LIN {X 0,Y 496.38,Z 733.448,A -85,B 0,C 180,E1 23641.747,E2 23641.747} C_VEL
LIN {X 0,Y 498.1,Z 714.982,A -85,B 0,C 180,E1 23640.21,E2 23640.21} C_VEL
LIN {X 0,Y 499.843,Z 694.815,A -85,B 0,C 180,E1 23638.795,E2 23638.795} C_VEL
LIN {X 0,Y 501.44,Z 674.409,A -85,B 0,C 180,E1 23637.63,E2 23637.63} C_VEL
LIN {X 0,Y 502.74,Z 652.978,A -85,B 0,C 180,E1 23636.672,E2 23636.672} C_VEL
LIN {X 0,Y 503.931,Z 629.73,A -85,B 0,C 180,E1 23635.874,E2 23635.874} C_VEL
LIN {X 0,Y 504.846,Z 606.635,A -85,B 0,C 180,E1 23635.308,E2 23635.308} C_VEL
LIN {X 0,Y 505.722,Z 566.306,A -85,B 0,C 180,E1 23634.669,E2 23634.669} C_VEL
LIN {X 0,Y 510.163,Z 554.646,A -85,B 0,C 180,E1 23634.04,E2 23634.04} C_VEL
LIN {X 0,Y 517.035,Z 539.66,A -85,B 0,C 180,E1 23633.305,E2 23633.305} C_VEL
LIN {X 0,Y 524.488,Z 527.632,A -85,B 0,C 180,E1 23632.83,E2 23632.83} C_VEL
LIN {X 0,Y 526.737,Z 523.652,A -85,B 0,C 180,E1 23632.664,E2 23632.664} C_VEL
LIN {X 0,Y 533.302,Z 512.044,A -85,B 0,C 180,E1 23632.187,E2 23632.187} C_VEL
LIN {X 0,Y 542.453,Z 498.435,A -85,B 0,C 180,E1 23631.8,E2 23631.8} C_VEL
LIN {X 0,Y 552.676,Z 482.618,A -85,B 0,C 180,E1 23631.568,E2 23631.568} C_VEL
LIN {X 0,Y 561.127,Z 466.92,A -85,B 0,C 180,E1 23631.466,E2 23631.466} C_VEL
LIN {X 0,Y 567.26,Z 452.489,A -85,B 0,C 180,E1 23631.429,E2 23631.429} C_VEL
LIN {X 0,Y 565.896,Z 454.329,A -85,B 0,C 180,E1 23630.864,E2 23630.864} C_VEL
LIN {X 0,Y 563.058,Z 455.358,A -85,B 0,C 180,E1 23630.255,E2 23630.255} C_VEL
LIN {X 0,Y 559.403,Z 455.291,A -85,B 0,C 180,E1 23629.747,E2 23629.747} C_VEL
LIN {X 0,Y 554.286,Z 453.945,A -85,B 0,C 180,E1 23629.255,E2 23629.255} C_VEL
LIN {X 0,Y 543.774,Z 449.42,A -85,B 0,C 180,E1 23628.29,E2 23628.29} C_VEL
LIN {X 0,Y 534.055,Z 443.361,A -85,B 0,C 180,E1 23627.214,E2 23627.214} C_VEL
LIN {X 0,Y 525.272,Z 435.554,A -85,B 0,C 180,E1 23626.015,E2 23626.015} C_VEL
LIN {X 0,Y 517.9,Z 426.094,A -85,B 0,C 180,E1 23624.727,E2 23624.727} C_VEL
LIN {X 0,Y 512.311,Z 415.203,A -85,B 0,C 180,E1 23623.392,E2 23623.392} C_VEL
LIN {X 0,Y 508.641,Z 403.465,A -85,B 0,C 180,E1 23622.091,E2 23622.091} C_VEL
LIN {X 0,Y 506.405,Z 389.242,A -85,B 0,C 180,E1 23620.659,E2 23620.659} C_VEL
LIN {X 0,Y 505.979,Z 373.52,A -85,B 0,C 180,E1 23619.223,E2 23619.223} C_VEL
LIN {X 0,Y 509.789,Z 322.987,A -85,B 0,C 180,E1 23614.931,E2 23614.931} C_VEL
LIN {X 0,Y 511.824,Z 299.18,A -85,B 0,C 180,E1 23612.833,E2 23612.833} C_VEL
LIN {X 0,Y 504.534,Z 283.166,A -85,B 0,C 180,E1 23610.222,E2 23610.222} C_VEL
LIN {X 0,Y 500.176,Z 274.319,A -85,B 0,C 180,E1 23608.628,E2 23608.628} C_VEL
LIN {X 0,Y 497.624,Z 274.818,A -85,B 0,C 180,E1 23608.306,E2 23608.306} C_VEL
LIN {X 0,Y 495.141,Z 275.99,A -85,B 0,C 180,E1 23608.067,E2 23608.067} C_VEL
LIN {X 0,Y 493.25,Z 276.086,A -85,B 0,C 180,E1 23607.789,E2 23607.789} C_VEL
LIN {X 0,Y 492.541,Z 275.81,A -85,B 0,C 180,E1 23607.619,E2 23607.619} C_VEL
LIN {X 0,Y 493.172,Z 322.85,A -85,B 0,C 180,E1 23604.558,E2 23604.558} C_VEL
LIN {X 0,Y 493.39,Z 364.566,A -85,B 0,C 180,E1 23601.705,E2 23601.705} C_VEL
LIN {X 0,Y 493.167,Z 403.632,A -85,B 0,C 180,E1 23598.928,E2 23598.928} C_VEL
LIN {X 0,Y 492.679,Z 449.513,A -85,B 0,C 180,E1 23595.598,E2 23595.598} C_VEL
LIN {X 0,Y 491.957,Z 495.066,A -85,B 0,C 180,E1 23592.202,E2 23592.202} C_VEL
LIN {X 0,Y 491.446,Z 499.514,A -85,B 0,C 180,E1 23591.926,E2 23591.926} C_VEL
LIN {X 0,Y 490.668,Z 612.915,A -85,B 0,C 180,E1 23590.126,E2 23590.126} C_VEL
LIN {X 0,Y 490.606,Z 628.131,A -85,B 0,C 180,E1 23589.649,E2 23589.649} C_VEL
LIN {X 0,Y 490.477,Z 641.255,A -85,B 0,C 180,E1 23589.031,E2 23589.031} C_VEL
LIN {X 0,Y 490.233,Z 654.167,A -85,B 0,C 180,E1 23588.208,E2 23588.208} C_VEL
LIN {X 0,Y 489.961,Z 666.706,A -85,B 0,C 180,E1 23587.15,E2 23587.15} C_VEL
LIN {X 0,Y 489.656,Z 677.457,A -85,B 0,C 180,E1 23585.977,E2 23585.977} C_VEL
LIN {X 0,Y 489.379,Z 686.759,A -85,B 0,C 180,E1 23584.687,E2 23584.687} C_VEL
LIN {X 0,Y 489.133,Z 694.688,A -85,B 0,C 180,E1 23583.281,E2 23583.281} C_VEL
LIN {X 0,Y 488.904,Z 701.596,A -85,B 0,C 180,E1 23581.64,E2 23581.64} C_VEL
LIN {X 0,Y 488.763,Z 706.452,A -85,B 0,C 180,E1 23580,E2 23580} C_VEL
LIN {X 0,Y 488.665,Z 709.537,A -85,B 0,C 180,E1 23578.358,E2 23578.358} C_VEL
LIN {X 0,Y 488.621,Z 711,A -85,B 0,C 180,E1 23576.598,E2 23576.598} C_VEL
LIN {X 0,Y 488.594,Z 710.599,A -85,B 0,C 180,E1 23574.834,E2 23574.834} C_VEL
LIN {X 0,Y 488.619,Z 708.56,A -85,B 0,C 180,E1 23573.183,E2 23573.183} C_VEL
LIN {X 0,Y 488.682,Z 704.854,A -85,B 0,C 180,E1 23571.528,E2 23571.528} C_VEL
LIN {X 0,Y 488.813,Z 699.231,A -85,B 0,C 180,E1 23569.868,E2 23569.868} C_VEL
LIN {X 0,Y 489.009,Z 692.043,A -85,B 0,C 180,E1 23568.321,E2 23568.321} C_VEL
LIN {X 0,Y 489.261,Z 683.364,A -85,B 0,C 180,E1 23566.888,E2 23566.888} C_VEL
LIN {X 0,Y 489.573,Z 673.151,A -85,B 0,C 180,E1 23565.572,E2 23565.572} C_VEL
LIN {X 0,Y 489.896,Z 661.171,A -85,B 0,C 180,E1 23564.371,E2 23564.371} C_VEL
LIN {X 0,Y 490.193,Z 648.737,A -85,B 0,C 180,E1 23563.407,E2 23563.407} C_VEL
LIN {X 0,Y 490.459,Z 635.31,A -85,B 0,C 180,E1 23562.616,E2 23562.616} C_VEL
LIN {X 0,Y 490.638,Z 620.571,A -85,B 0,C 180,E1 23561.997,E2 23561.997} C_VEL
LIN {X 0,Y 490.728,Z 604.678,A -85,B 0,C 180,E1 23561.586,E2 23561.586} C_VEL
LIN {X 0,Y 491.469,Z 494.156,A -85,B 0,C 180,E1 23559.859,E2 23559.859} C_VEL
LIN {X 0,Y 492.377,Z 448.014,A -85,B 0,C 180,E1 23556.326,E2 23556.326} C_VEL
LIN {X 0,Y 493.343,Z 402.982,A -85,B 0,C 180,E1 23552.87,E2 23552.87} C_VEL
LIN {X 0,Y 494.194,Z 357.923,A -85,B 0,C 180,E1 23549.413,E2 23549.413} C_VEL
LIN {X 0,Y 494.758,Z 323.358,A -85,B 0,C 180,E1 23546.764,E2 23546.764} C_VEL
LIN {X 0,Y 493.985,Z 317.131,A -85,B 0,C 180,E1 23546.234,E2 23546.234} C_VEL
LIN {X 0,Y 488.35,Z 301.373,A -85,B 0,C 180,E1 23544.701,E2 23544.701} C_VEL
LIN {X 0,Y 487.701,Z 295.968,A -85,B 0,C 180,E1 23544.249,E2 23544.249} C_VEL
LIN {X 0,Y 488.094,Z 275.29,A -85,B 0,C 180,E1 23542.639,E2 23542.639} C_VEL
LIN {X 0,Y 480.862,Z 252.836,A -85,B 0,C 180,E1 23540.451,E2 23540.451} C_VEL
LIN {X 0,Y 480.895,Z 253.018,A -85,B 0,C 180,E1 23539.085,E2 23539.085} C_VEL
LIN {X 0,Y 482.364,Z 256.557,A -85,B 0,C 180,E1 23538.265,E2 23538.265} C_VEL
LIN {X 0,Y 483.282,Z 257.796,A -85,B 0,C 180,E1 23537.907,E2 23537.907} C_VEL
LIN {X 0,Y 485.144,Z 261.755,A -85,B 0,C 180,E1 23536.985,E2 23536.985} C_VEL
LIN {X 0,Y 490.291,Z 272.658,A -85,B 0,C 180,E1 23534.55,E2 23534.55} C_VEL
LIN {X 0,Y 495.139,Z 283.311,A -85,B 0,C 180,E1 23532.346,E2 23532.346} C_VEL
LIN {X 0,Y 500.066,Z 295.346,A -85,B 0,C 180,E1 23530.078,E2 23530.078} C_VEL
LIN {X 0,Y 497.632,Z 318.632,A -85,B 0,C 180,E1 23527.59,E2 23527.59} C_VEL
LIN {X 0,Y 498.99,Z 325.374,A -85,B 0,C 180,E1 23527.35,E2 23527.35} C_VEL
LIN {X 0,Y 496.803,Z 427.751,A -85,B 0,C 180,E1 23525.65,E2 23525.65} C_VEL
LIN {X 0,Y 493.178,Z 568.271,A -85,B 0,C 180,E1 23523.126,E2 23523.126} C_VEL
LIN {X 0,Y 492.401,Z 589.199,A -85,B 0,C 180,E1 23522.533,E2 23522.533} C_VEL
LIN {X 0,Y 491.403,Z 608.833,A -85,B 0,C 180,E1 23521.761,E2 23521.761} C_VEL
LIN {X 0,Y 490.219,Z 627.883,A -85,B 0,C 180,E1 23520.794,E2 23520.794} C_VEL
LIN {X 0,Y 488.842,Z 646.705,A -85,B 0,C 180,E1 23519.601,E2 23519.601} C_VEL
LIN {X 0,Y 487.423,Z 664.686,A -85,B 0,C 180,E1 23518.208,E2 23518.208} C_VEL
LIN {X 0,Y 485.977,Z 681.431,A -85,B 0,C 180,E1 23516.649,E2 23516.649} C_VEL
LIN {X 0,Y 484.672,Z 696.234,A -85,B 0,C 180,E1 23515.018,E2 23515.018} C_VEL
LIN {X 0,Y 483.407,Z 710.599,A -85,B 0,C 180,E1 23513.141,E2 23513.141} C_VEL
LIN {X 0,Y 482.297,Z 723.641,A -85,B 0,C 180,E1 23511.106,E2 23511.106} C_VEL
LIN {X 0,Y 481.388,Z 735.453,A -85,B 0,C 180,E1 23508.906,E2 23508.906} C_VEL
LIN {X 0,Y 480.799,Z 744.274,A -85,B 0,C 180,E1 23506.926,E2 23506.926} C_VEL
LIN {X 0,Y 480.356,Z 753.265,A -85,B 0,C 180,E1 23504.588,E2 23504.588} C_VEL
LIN {X 0,Y 480.101,Z 760.219,A -85,B 0,C 180,E1 23502.265,E2 23502.265} C_VEL
LIN {X 0,Y 479.985,Z 765.081,A -85,B 0,C 180,E1 23500.199,E2 23500.199} C_VEL
LIN {X 0,Y 479.931,Z 769.255,A -85,B 0,C 180,E1 23497.783,E2 23497.783} C_VEL
LIN {X 0,Y 479.905,Z 771.524,A -85,B 0,C 180,E1 23495.5,E2 23495.5} C_VEL
LIN {X 0,Y 479.903,Z 772.375,A -85,B 0,C 180,E1 23493.464,E2 23493.464} C_VEL
LIN {X 0,Y 479.907,Z 772.03,A -85,B 0,C 180,E1 23491.194,E2 23491.194} C_VEL
LIN {X 0,Y 479.913,Z 769.901,A -85,B 0,C 180,E1 23488.687,E2 23488.687} C_VEL
LIN {X 0,Y 479.948,Z 766.881,A -85,B 0,C 180,E1 23486.656,E2 23486.656} C_VEL
LIN {X 0,Y 480.034,Z 762.684,A -85,B 0,C 180,E1 23484.622,E2 23484.622} C_VEL
LIN {X 0,Y 480.242,Z 756.178,A -85,B 0,C 180,E1 23482.222,E2 23482.222} C_VEL
LIN {X 0,Y 480.57,Z 748.581,A -85,B 0,C 180,E1 23480.056,E2 23480.056} C_VEL
LIN {X 0,Y 481.199,Z 738.233,A -85,B 0,C 180,E1 23477.58,E2 23477.58} C_VEL
LIN {X 0,Y 481.993,Z 727.382,A -85,B 0,C 180,E1 23475.463,E2 23475.463} C_VEL
LIN {X 0,Y 483.026,Z 714.869,A -85,B 0,C 180,E1 23473.402,E2 23473.402} C_VEL
LIN {X 0,Y 484.264,Z 700.8,A -85,B 0,C 180,E1 23471.46,E2 23471.46} C_VEL
LIN {X 0,Y 485.557,Z 686.249,A -85,B 0,C 180,E1 23469.76,E2 23469.76} C_VEL
LIN {X 0,Y 487.016,Z 669.572,A -85,B 0,C 180,E1 23468.122,E2 23468.122} C_VEL
LIN {X 0,Y 488.472,Z 651.962,A -85,B 0,C 180,E1 23466.683,E2 23466.683} C_VEL
LIN {X 0,Y 489.911,Z 632.774,A -85,B 0,C 180,E1 23465.396,E2 23465.396} C_VEL
LIN {X 0,Y 491.095,Z 614.617,A -85,B 0,C 180,E1 23464.415,E2 23464.415} C_VEL
LIN {X 0,Y 492.12,Z 595.098,A -85,B 0,C 180,E1 23463.584,E2 23463.584} C_VEL
LIN {X 0,Y 492.975,Z 574.762,A -85,B 0,C 180,E1 23462.943,E2 23462.943} C_VEL
LIN {X 0,Y 493.591,Z 552.537,A -85,B 0,C 180,E1 23462.471,E2 23462.471} C_VEL
LIN {X 0,Y 497.835,Z 385.617,A -85,B 0,C 180,E1 23459.542,E2 23459.542} C_VEL
LIN {X 0,Y 498.921,Z 320.717,A -85,B 0,C 180,E1 23458.474,E2 23458.474} C_VEL
LIN {X 0,Y 498.1,Z 316.099,A -85,B 0,C 180,E1 23458.303,E2 23458.303} C_VEL
LIN {X 0,Y 500.032,Z 293.482,A -85,B 0,C 180,E1 23456.288,E2 23456.288} C_VEL
LIN {X 0,Y 492.25,Z 276.567,A -85,B 0,C 180,E1 23453.549,E2 23453.549} C_VEL
LIN {X 0,Y 486.502,Z 264.754,A -85,B 0,C 180,E1 23451.484,E2 23451.484} C_VEL
LIN {X 0,Y 484.789,Z 261.244,A -85,B 0,C 180,E1 23450.85,E2 23450.85} C_VEL
LIN {X 0,Y 482.59,Z 256.865,A -85,B 0,C 180,E1 23450.038,E2 23450.038} C_VEL
LIN {X 0,Y 480.993,Z 253.436,A -85,B 0,C 180,E1 23449.409,E2 23449.409} C_VEL
LIN {X 0,Y 480.894,Z 252.838,A -85,B 0,C 180,E1 23449.321,E2 23449.321} C_VEL
LIN {X 0,Y 480.885,Z 252.835,A -85,B 0,C 180,E1 23445.664,E2 23445.664} C_VEL
LIN {X 0,Y 480.883,Z 252.833,A -85,B 0,C 180,E1 23442.03,E2 23442.03} C_VEL
LIN {X 0,Y 480.896,Z 252.833,A -85,B 0,C 180,E1 23438.386,E2 23438.386} C_VEL
LIN {X 0,Y 480.882,Z 252.837,A -85,B 0,C 180,E1 23434.73,E2 23434.73} C_VEL
LIN {X 0,Y 480.882,Z 252.884,A -85,B 0,C 180,E1 23431.161,E2 23431.161} C_VEL
LIN {X 0,Y 488.38,Z 276.554,A -85,B 0,C 180,E1 23428.692,E2 23428.692} C_VEL
LIN {X 0,Y 487.688,Z 321.036,A -85,B 0,C 180,E1 23424.983,E2 23424.983} C_VEL
LIN {X 0,Y 486.877,Z 362.038,A -85,B 0,C 180,E1 23421.568,E2 23421.568} C_VEL
LIN {X 0,Y 485.897,Z 404.107,A -85,B 0,C 180,E1 23418.067,E2 23418.067} C_VEL
LIN {X 0,Y 484.975,Z 446.252,A -85,B 0,C 180,E1 23414.587,E2 23414.587} C_VEL
LIN {X 0,Y 485.216,Z 454.797,A -85,B 0,C 180,E1 23414.435,E2 23414.435} C_VEL
LIN {X 0,Y 483.933,Z 589.379,A -85,B 0,C 180,E1 23412.267,E2 23412.267} C_VEL
LIN {X 0,Y 483.783,Z 605.964,A -85,B 0,C 180,E1 23411.777,E2 23411.777} C_VEL
LIN {X 0,Y 483.477,Z 621.487,A -85,B 0,C 180,E1 23411.089,E2 23411.089} C_VEL
LIN {X 0,Y 483.104,Z 636.557,A -85,B 0,C 180,E1 23410.193,E2 23410.193} C_VEL
LIN {X 0,Y 482.632,Z 651.077,A -85,B 0,C 180,E1 23409.059,E2 23409.059} C_VEL
LIN {X 0,Y 482.198,Z 663.25,A -85,B 0,C 180,E1 23407.866,E2 23407.866} C_VEL
LIN {X 0,Y 481.749,Z 674.924,A -85,B 0,C 180,E1 23406.435,E2 23406.435} C_VEL
LIN {X 0,Y 481.367,Z 685.044,A -85,B 0,C 180,E1 23404.886,E2 23404.886} C_VEL
LIN {X 0,Y 481.07,Z 693.633,A -85,B 0,C 180,E1 23403.217,E2 23403.217} C_VEL
LIN {X 0,Y 480.885,Z 700.29,A -85,B 0,C 180,E1 23401.549,E2 23401.549} C_VEL
LIN {X 0,Y 480.74,Z 705.866,A -85,B 0,C 180,E1 23399.643,E2 23399.643} C_VEL
LIN {X 0,Y 480.686,Z 709.337,A -85,B 0,C 180,E1 23397.855,E2 23397.855} C_VEL
LIN {X 0,Y 480.667,Z 711.381,A -85,B 0,C 180,E1 23395.825,E2 23395.825} C_VEL
LIN {X 0,Y 480.706,Z 711.456,A -85,B 0,C 180,E1 23393.911,E2 23393.911} C_VEL
LIN {X 0,Y 480.777,Z 709.805,A -85,B 0,C 180,E1 23391.991,E2 23391.991} C_VEL
LIN {X 0,Y 480.905,Z 706.23,A -85,B 0,C 180,E1 23390.063,E2 23390.063} C_VEL
LIN {X 0,Y 481.093,Z 701.074,A -85,B 0,C 180,E1 23388.249,E2 23388.249} C_VEL
LIN {X 0,Y 481.341,Z 693.803,A -85,B 0,C 180,E1 23386.425,E2 23386.425} C_VEL
LIN {X 0,Y 481.666,Z 685.525,A -85,B 0,C 180,E1 23384.838,E2 23384.838} C_VEL
LIN {X 0,Y 482.074,Z 674.914,A -85,B 0,C 180,E1 23383.244,E2 23383.244} C_VEL
LIN {X 0,Y 482.486,Z 663.45,A -85,B 0,C 180,E1 23381.89,E2 23381.89} C_VEL
LIN {X 0,Y 482.88,Z 651.01,A -85,B 0,C 180,E1 23380.716,E2 23380.716} C_VEL
LIN {X 0,Y 483.211,Z 637.613,A -85,B 0,C 180,E1 23379.721,E2 23379.721} C_VEL
LIN {X 0,Y 483.487,Z 622.444,A -85,B 0,C 180,E1 23378.857,E2 23378.857} C_VEL
LIN {X 0,Y 483.652,Z 606.109,A -85,B 0,C 180,E1 23378.197,E2 23378.197} C_VEL
LIN {X 0,Y 483.672,Z 589.924,A -85,B 0,C 180,E1 23377.774,E2 23377.774} C_VEL
LIN {X 0,Y 484.709,Z 473.284,A -85,B 0,C 180,E1 23375.896,E2 23375.896} C_VEL
LIN {X 0,Y 485.05,Z 452.809,A -85,B 0,C 180,E1 23375.523,E2 23375.523} C_VEL
LIN {X 0,Y 485.709,Z 447.24,A -85,B 0,C 180,E1 23375.104,E2 23375.104} C_VEL
LIN {X 0,Y 486.235,Z 406.579,A -85,B 0,C 180,E1 23371.906,E2 23371.906} C_VEL
LIN {X 0,Y 486.403,Z 373.966,A -85,B 0,C 180,E1 23369.426,E2 23369.426} C_VEL
LIN {X 0,Y 486.241,Z 335.387,A -85,B 0,C 180,E1 23366.602,E2 23366.602} C_VEL
LIN {X 0,Y 486.068,Z 315.437,A -85,B 0,C 180,E1 23365.175,E2 23365.175} C_VEL
LIN {X 0,Y 487.432,Z 316.242,A -85,B 0,C 180,E1 23364.946,E2 23364.946} C_VEL
LIN {X 0,Y 489.679,Z 316.055,A -85,B 0,C 180,E1 23364.701,E2 23364.701} C_VEL
LIN {X 0,Y 491.846,Z 315.218,A -85,B 0,C 180,E1 23364.523,E2 23364.523} C_VEL
LIN {X 0,Y 495.198,Z 315.029,A -85,B 0,C 180,E1 23364.159,E2 23364.159} C_VEL
LIN {X 0,Y 498.446,Z 314.267,A -85,B 0,C 180,E1 23363.861,E2 23363.861} C_VEL
LIN {X 0,Y 503.576,Z 313.442,A -85,B 0,C 180,E1 23363.37,E2 23363.37} C_VEL
LIN {X 0,Y 502.225,Z 340.421,A -85,B 0,C 180,E1 23361.382,E2 23361.382} C_VEL
LIN {X 0,Y 503.133,Z 357.34,A -85,B 0,C 180,E1 23359.994,E2 23359.994} C_VEL
LIN {X 0,Y 505.646,Z 371.909,A -85,B 0,C 180,E1 23358.666,E2 23358.666} C_VEL
LIN {X 0,Y 509.605,Z 384.438,A -85,B 0,C 180,E1 23357.399,E2 23357.399} C_VEL
LIN {X 0,Y 515.13,Z 395.571,A -85,B 0,C 180,E1 23356.138,E2 23356.138} C_VEL
LIN {X 0,Y 522.184,Z 405.312,A -85,B 0,C 180,E1 23354.891,E2 23354.891} C_VEL
LIN {X 0,Y 530.1,Z 413.14,A -85,B 0,C 180,E1 23353.747,E2 23353.747} C_VEL
LIN {X 0,Y 540.174,Z 420.213,A -85,B 0,C 180,E1 23352.55,E2 23352.55} C_VEL
LIN {X 0,Y 551.135,Z 425.486,A -85,B 0,C 180,E1 23351.466,E2 23351.466} C_VEL
LIN {X 0,Y 560.238,Z 428.38,A -85,B 0,C 180,E1 23350.668,E2 23350.668} C_VEL
LIN {X 0,Y 564.412,Z 428.784,A -85,B 0,C 180,E1 23350.153,E2 23350.153} C_VEL
LIN {X 0,Y 566.541,Z 428.672,A -85,B 0,C 180,E1 23349.758,E2 23349.758} C_VEL
LIN {X 0,Y 564.158,Z 434.639,A -85,B 0,C 180,E1 23349.612,E2 23349.612} C_VEL
LIN {X 0,Y 554.295,Z 452.798,A -85,B 0,C 180,E1 23349.463,E2 23349.463} C_VEL
LIN {X 0,Y 542.754,Z 471.192,A -85,B 0,C 180,E1 23349.144,E2 23349.144} C_VEL
LIN {X 0,Y 529.479,Z 492.499,A -85,B 0,C 180,E1 23348.617,E2 23348.617} C_VEL
LIN {X 0,Y 521.442,Z 507.86,A -85,B 0,C 180,E1 23348.129,E2 23348.129} C_VEL
LIN {X 0,Y 516.353,Z 520.01,A -85,B 0,C 180,E1 23347.657,E2 23347.657} C_VEL
LIN {X 0,Y 509.506,Z 533.706,A -85,B 0,C 180,E1 23347.181,E2 23347.181} C_VEL
LIN {X 0,Y 504.963,Z 545.921,A -85,B 0,C 180,E1 23346.655,E2 23346.655} C_VEL
LIN {X 0,Y 500.019,Z 560.23,A -85,B 0,C 180,E1 23346.008,E2 23346.008} C_VEL
LIN {X 0,Y 499.1,Z 563.948,A -85,B 0,C 180,E1 23345.861,E2 23345.861} C_VEL
LIN {X 0,Y 498.399,Z 593.728,A -85,B 0,C 180,E1 23345.409,E2 23345.409} C_VEL
LIN {X 0,Y 497.549,Z 617.702,A -85,B 0,C 180,E1 23344.92,E2 23344.92} C_VEL
LIN {X 0,Y 496.401,Z 640.592,A -85,B 0,C 180,E1 23344.236,E2 23344.236} C_VEL
LIN {X 0,Y 495.064,Z 662.664,A -85,B 0,C 180,E1 23343.357,E2 23343.357} C_VEL
LIN {X 0,Y 493.532,Z 684.32,A -85,B 0,C 180,E1 23342.265,E2 23342.265} C_VEL
LIN {X 0,Y 491.889,Z 704.756,A -85,B 0,C 180,E1 23340.997,E2 23340.997} C_VEL
LIN {X 0,Y 490.417,Z 721.095,A -85,B 0,C 180,E1 23339.783,E2 23339.783} C_VEL
LIN {X 0,Y 488.503,Z 740.079,A -85,B 0,C 180,E1 23338.084,E2 23338.084} C_VEL
LIN {X 0,Y 486.678,Z 757.864,A -85,B 0,C 180,E1 23336.213,E2 23336.213} C_VEL
LIN {X 0,Y 484.943,Z 774.948,A -85,B 0,C 180,E1 23334.094,E2 23334.094} C_VEL
LIN {X 0,Y 483.4,Z 791.073,A -85,B 0,C 180,E1 23331.731,E2 23331.731} C_VEL
LIN {X 0,Y 482.171,Z 805.314,A -85,B 0,C 180,E1 23329.251,E2 23329.251} C_VEL
LIN {X 0,Y 481.256,Z 817.549,A -85,B 0,C 180,E1 23326.711,E2 23326.711} C_VEL
LIN {X 0,Y 480.623,Z 827.996,A -85,B 0,C 180,E1 23324.087,E2 23324.087} C_VEL
LIN {X 0,Y 480.228,Z 836.573,A -85,B 0,C 180,E1 23321.408,E2 23321.408} C_VEL
LIN {X 0,Y 480.015,Z 843.196,A -85,B 0,C 180,E1 23318.746,E2 23318.746} C_VEL
LIN {X 0,Y 479.938,Z 847.807,A -85,B 0,C 180,E1 23316.219,E2 23316.219} C_VEL
LIN {X 0,Y 479.909,Z 850.87,A -85,B 0,C 180,E1 23313.661,E2 23313.661} C_VEL
LIN {X 0,Y 479.91,Z 852.372,A -85,B 0,C 180,E1 23310.955,E2 23310.955} C_VEL
LIN {X 0,Y 479.899,Z 852.152,A -85,B 0,C 180,E1 23308.328,E2 23308.328} C_VEL
LIN {X 0,Y 479.915,Z 850.371,A -85,B 0,C 180,E1 23305.818,E2 23305.818} C_VEL
LIN {X 0,Y 479.957,Z 846.849,A -85,B 0,C 180,E1 23303.18,E2 23303.18} C_VEL
LIN {X 0,Y 480.072,Z 841.593,A -85,B 0,C 180,E1 23300.53,E2 23300.53} C_VEL
LIN {X 0,Y 480.31,Z 834.427,A -85,B 0,C 180,E1 23297.863,E2 23297.863} C_VEL
LIN {X 0,Y 480.752,Z 825.57,A -85,B 0,C 180,E1 23295.261,E2 23295.261} C_VEL
LIN {X 0,Y 481.437,Z 815,A -85,B 0,C 180,E1 23292.723,E2 23292.723} C_VEL
LIN {X 0,Y 482.332,Z 803.331,A -85,B 0,C 180,E1 23290.377,E2 23290.377} C_VEL
LIN {X 0,Y 483.473,Z 790.295,A -85,B 0,C 180,E1 23288.145,E2 23288.145} C_VEL
LIN {X 0,Y 484.988,Z 774.48,A -85,B 0,C 180,E1 23285.843,E2 23285.843} C_VEL
LIN {X 0,Y 486.71,Z 757.504,A -85,B 0,C 180,E1 23283.746,E2 23283.746} C_VEL
LIN {X 0,Y 488.565,Z 739.511,A -85,B 0,C 180,E1 23281.86,E2 23281.86} C_VEL
LIN {X 0,Y 490.417,Z 721.096,A -85,B 0,C 180,E1 23280.217,E2 23280.217} C_VEL
LIN {X 0,Y 491.89,Z 704.76,A -85,B 0,C 180,E1 23279.003,E2 23279.003} C_VEL
LIN {X 0,Y 493.523,Z 684.24,A -85,B 0,C 180,E1 23277.734,E2 23277.734} C_VEL
LIN {X 0,Y 495.105,Z 661.858,A -85,B 0,C 180,E1 23276.611,E2 23276.611} C_VEL
LIN {X 0,Y 496.481,Z 638.809,A -85,B 0,C 180,E1 23275.705,E2 23275.705} C_VEL
LIN {X 0,Y 497.615,Z 615.774,A -85,B 0,C 180,E1 23275.04,E2 23275.04} C_VEL
LIN {X 0,Y 498.381,Z 592.976,A -85,B 0,C 180,E1 23274.585,E2 23274.585} C_VEL
LIN {X 0,Y 499.034,Z 565.629,A -85,B 0,C 180,E1 23274.171,E2 23274.171} C_VEL
LIN {X 0,Y 499.312,Z 563.71,A -85,B 0,C 180,E1 23274.145,E2 23274.145} C_VEL
LIN {X 0,Y 503.862,Z 552.303,A -85,B 0,C 180,E1 23273.535,E2 23273.535} C_VEL
LIN {X 0,Y 510.541,Z 537.864,A -85,B 0,C 180,E1 23272.824,E2 23272.824} C_VEL
LIN {X 0,Y 517.954,Z 525.867,A -85,B 0,C 180,E1 23272.347,E2 23272.347} C_VEL
LIN {X 0,Y 520.245,Z 521.945,A -85,B 0,C 180,E1 23272.187,E2 23272.187} C_VEL
LIN {X 0,Y 526.825,Z 510.336,A -85,B 0,C 180,E1 23271.708,E2 23271.708} C_VEL
LIN {X 0,Y 536.729,Z 496.264,A -85,B 0,C 180,E1 23271.249,E2 23271.249} C_VEL
LIN {X 0,Y 549.126,Z 480.047,A -85,B 0,C 180,E1 23270.865,E2 23270.865} C_VEL
LIN {X 0,Y 559.176,Z 465.05,A -85,B 0,C 180,E1 23270.688,E2 23270.688} C_VEL
LIN {X 0,Y 560.818,Z 462.177,A -85,B 0,C 180,E1 23270.652,E2 23270.652} C_VEL
LIN {X 0,Y 556.708,Z 462.22,A -85,B 0,C 180,E1 23270.076,E2 23270.076} C_VEL
LIN {X 0,Y 551.539,Z 460.939,A -85,B 0,C 180,E1 23269.587,E2 23269.587} C_VEL
LIN {X 0,Y 540.155,Z 456.256,A -85,B 0,C 180,E1 23268.562,E2 23268.562} C_VEL
LIN {X 0,Y 529.628,Z 449.931,A -85,B 0,C 180,E1 23267.414,E2 23267.414} C_VEL
LIN {X 0,Y 520.709,Z 442.355,A -85,B 0,C 180,E1 23266.219,E2 23266.219} C_VEL
LIN {X 0,Y 512.885,Z 432.876,A -85,B 0,C 180,E1 23264.887,E2 23264.887} C_VEL
LIN {X 0,Y 507.27,Z 422.944,A -85,B 0,C 180,E1 23263.619,E2 23263.619} C_VEL
LIN {X 0,Y 503.046,Z 411.454,A -85,B 0,C 180,E1 23262.284,E2 23262.284} C_VEL
LIN {X 0,Y 500.267,Z 397.472,A -85,B 0,C 180,E1 23260.81,E2 23260.81} C_VEL
LIN {X 0,Y 499.292,Z 382.036,A -85,B 0,C 180,E1 23259.331,E2 23259.331} C_VEL
LIN {X 0,Y 500.645,Z 357.876,A -85,B 0,C 180,E1 23257.238,E2 23257.238} C_VEL
LIN {X 0,Y 504.106,Z 318.983,A -85,B 0,C 180,E1 23253.872,E2 23253.872} C_VEL
LIN {X 0,Y 505.57,Z 303.35,A -85,B 0,C 180,E1 23252.475,E2 23252.475} C_VEL
LIN {X 0,Y 498.672,Z 288.161,A -85,B 0,C 180,E1 23249.95,E2 23249.95} C_VEL
LIN {X 0,Y 495.465,Z 281.71,A -85,B 0,C 180,E1 23248.77,E2 23248.77} C_VEL
LIN {X 0,Y 492.031,Z 282.889,A -85,B 0,C 180,E1 23248.392,E2 23248.392} C_VEL
LIN {X 0,Y 490.315,Z 283.206,A -85,B 0,C 180,E1 23248.169,E2 23248.169} C_VEL
LIN {X 0,Y 487.449,Z 284.527,A -85,B 0,C 180,E1 23247.883,E2 23247.883} C_VEL
LIN {X 0,Y 485.632,Z 284.494,A -85,B 0,C 180,E1 23247.596,E2 23247.596} C_VEL
LIN {X 0,Y 485.142,Z 284.235,A -85,B 0,C 180,E1 23247.477,E2 23247.477} C_VEL
LIN {X 0,Y 485.749,Z 328.431,A -85,B 0,C 180,E1 23244.569,E2 23244.569} C_VEL
LIN {X 0,Y 485.861,Z 371.281,A -85,B 0,C 180,E1 23241.614,E2 23241.614} C_VEL
LIN {X 0,Y 485.548,Z 419.344,A -85,B 0,C 180,E1 23238.178,E2 23238.178} C_VEL
LIN {X 0,Y 484.87,Z 466.154,A -85,B 0,C 180,E1 23234.728,E2 23234.728} C_VEL
LIN {X 0,Y 484.263,Z 497.232,A -85,B 0,C 180,E1 23232.399,E2 23232.399} C_VEL
LIN {X 0,Y 483.749,Z 501.19,A -85,B 0,C 180,E1 23232.163,E2 23232.163} C_VEL
LIN {X 0,Y 482.895,Z 614.459,A -85,B 0,C 180,E1 23230.317,E2 23230.317} C_VEL
LIN {X 0,Y 482.846,Z 629.57,A -85,B 0,C 180,E1 23229.836,E2 23229.836} C_VEL
LIN {X 0,Y 482.707,Z 643.257,A -85,B 0,C 180,E1 23229.177,E2 23229.177} C_VEL
LIN {X 0,Y 482.451,Z 656.435,A -85,B 0,C 180,E1 23228.31,E2 23228.31} C_VEL
LIN {X 0,Y 482.174,Z 668.503,A -85,B 0,C 180,E1 23227.267,E2 23227.267} C_VEL
LIN {X 0,Y 481.827,Z 680.148,A -85,B 0,C 180,E1 23225.955,E2 23225.955} C_VEL
LIN {X 0,Y 481.511,Z 689.887,A -85,B 0,C 180,E1 23224.525,E2 23224.525} C_VEL
LIN {X 0,Y 481.242,Z 697.391,A -85,B 0,C 180,E1 23223.096,E2 23223.096} C_VEL
LIN {X 0,Y 481.035,Z 703.565,A -85,B 0,C 180,E1 23221.548,E2 23221.548} C_VEL
LIN {X 0,Y 480.871,Z 708.507,A -85,B 0,C 180,E1 23219.761,E2 23219.761} C_VEL
LIN {X 0,Y 480.773,Z 711.389,A -85,B 0,C 180,E1 23217.973,E2 23217.973} C_VEL
LIN {X 0,Y 480.717,Z 712.383,A -85,B 0,C 180,E1 23216.183,E2 23216.183} C_VEL
LIN {X 0,Y 480.706,Z 711.653,A -85,B 0,C 180,E1 23214.509,E2 23214.509} C_VEL
LIN {X 0,Y 480.743,Z 709.057,A -85,B 0,C 180,E1 23212.711,E2 23212.711} C_VEL
LIN {X 0,Y 480.838,Z 704.447,A -85,B 0,C 180,E1 23210.907,E2 23210.907} C_VEL
LIN {X 0,Y 481.004,Z 698.083,A -85,B 0,C 180,E1 23209.217,E2 23209.217} C_VEL
LIN {X 0,Y 481.224,Z 690.77,A -85,B 0,C 180,E1 23207.764,E2 23207.764} C_VEL
LIN {X 0,Y 481.525,Z 681.309,A -85,B 0,C 180,E1 23206.307,E2 23206.307} C_VEL
LIN {X 0,Y 481.869,Z 670.1,A -85,B 0,C 180,E1 23204.967,E2 23204.967} C_VEL
LIN {X 0,Y 482.211,Z 657.531,A -85,B 0,C 180,E1 23203.806,E2 23203.806} C_VEL
LIN {X 0,Y 482.547,Z 643.518,A -85,B 0,C 180,E1 23202.826,E2 23202.826} C_VEL
LIN {X 0,Y 482.772,Z 629.023,A -85,B 0,C 180,E1 23202.089,E2 23202.089} C_VEL
LIN {X 0,Y 482.902,Z 614.383,A -85,B 0,C 180,E1 23201.585,E2 23201.585} C_VEL
LIN {X 0,Y 482.941,Z 597.395,A -85,B 0,C 180,E1 23201.255,E2 23201.255} C_VEL
LIN {X 0,Y 483.8,Z 495.19,A -85,B 0,C 180,E1 23199.62,E2 23199.62} C_VEL
LIN {X 0,Y 484.747,Z 449.326,A -85,B 0,C 180,E1 23196.089,E2 23196.089} C_VEL
LIN {X 0,Y 485.741,Z 405.082,A -85,B 0,C 180,E1 23192.675,E2 23192.675} C_VEL
LIN {X 0,Y 486.64,Z 360.415,A -85,B 0,C 180,E1 23189.229,E2 23189.229} C_VEL
LIN {X 0,Y 487.4,Z 316.937,A -85,B 0,C 180,E1 23185.87,E2 23185.87} C_VEL
LIN {X 0,Y 487.701,Z 295.968,A -85,B 0,C 180,E1 23184.249,E2 23184.249} C_VEL
LIN {X 0,Y 486.967,Z 289.679,A -85,B 0,C 180,E1 23183.712,E2 23183.712} C_VEL
LIN {X 0,Y 484.214,Z 282.304,A -85,B 0,C 180,E1 23182.966,E2 23182.966} C_VEL
LIN {X 0,Y 478.3,Z 270.271,A -85,B 0,C 180,E1 23181.697,E2 23181.697} C_VEL
LIN {X 0,Y 478.01,Z 269.419,A -85,B 0,C 180,E1 23181.613,E2 23181.613} C_VEL
LIN {X 0,Y 473.317,Z 255.454,A -85,B 0,C 180,E1 23180.202,E2 23180.202} C_VEL
LIN {X 0,Y 475.509,Z 259.245,A -85,B 0,C 180,E1 23179.16,E2 23179.16} C_VEL
LIN {X 0,Y 477.457,Z 263,A -85,B 0,C 180,E1 23178.204,E2 23178.204} C_VEL
LIN {X 0,Y 482.245,Z 273.051,A -85,B 0,C 180,E1 23175.839,E2 23175.839} C_VEL
LIN {X 0,Y 487.467,Z 284.194,A -85,B 0,C 180,E1 23173.404,E2 23173.404} C_VEL
LIN {X 0,Y 493.741,Z 299.324,A -85,B 0,C 180,E1 23170.454,E2 23170.454} C_VEL
LIN {X 0,Y 491.419,Z 320.977,A -85,B 0,C 180,E1 23168.115,E2 23168.115} C_VEL
LIN {X 0,Y 492.633,Z 327.035,A -85,B 0,C 180,E1 23167.893,E2 23167.893} C_VEL
LIN {X 0,Y 490.472,Z 421.582,A -85,B 0,C 180,E1 23166.303,E2 23166.303} C_VEL
LIN {X 0,Y 486.104,Z 569.119,A -85,B 0,C 180,E1 23163.554,E2 23163.554} C_VEL
LIN {X 0,Y 485.29,Z 589.615,A -85,B 0,C 180,E1 23162.962,E2 23162.962} C_VEL
LIN {X 0,Y 484.199,Z 609.905,A -85,B 0,C 180,E1 23162.151,E2 23162.151} C_VEL
LIN {X 0,Y 482.954,Z 628.884,A -85,B 0,C 180,E1 23161.17,E2 23161.17} C_VEL
LIN {X 0,Y 481.504,Z 647.666,A -85,B 0,C 180,E1 23159.961,E2 23159.961} C_VEL
LIN {X 0,Y 479.951,Z 666.263,A -85,B 0,C 180,E1 23158.494,E2 23158.494} C_VEL
LIN {X 0,Y 478.419,Z 682.975,A -85,B 0,C 180,E1 23156.902,E2 23156.902} C_VEL
LIN {X 0,Y 476.985,Z 698.152,A -85,B 0,C 180,E1 23155.184,E2 23155.184} C_VEL
LIN {X 0,Y 475.66,Z 712.377,A -85,B 0,C 180,E1 23153.277,E2 23153.277} C_VEL
LIN {X 0,Y 474.523,Z 725.128,A -85,B 0,C 180,E1 23151.249,E2 23151.249} C_VEL
LIN {X 0,Y 473.538,Z 736.983,A -85,B 0,C 180,E1 23148.976,E2 23148.976} C_VEL
LIN {X 0,Y 472.836,Z 746.827,A -85,B 0,C 180,E1 23146.68,E2 23146.68} C_VEL
LIN {X 0,Y 472.335,Z 755.352,A -85,B 0,C 180,E1 23144.215,E2 23144.215} C_VEL
LIN {X 0,Y 472.088,Z 761.423,A -85,B 0,C 180,E1 23141.98,E2 23141.98} C_VEL
LIN {X 0,Y 471.953,Z 767.071,A -85,B 0,C 180,E1 23139.266,E2 23139.266} C_VEL
LIN {X 0,Y 471.925,Z 770.148,A -85,B 0,C 180,E1 23137.059,E2 23137.059} C_VEL
LIN {X 0,Y 471.913,Z 771.946,A -85,B 0,C 180,E1 23134.862,E2 23134.862} C_VEL
LIN {X 0,Y 471.906,Z 772.356,A -85,B 0,C 180,E1 23132.186,E2 23132.186} C_VEL
LIN {X 0,Y 471.918,Z 771.238,A -85,B 0,C 180,E1 23130,E2 23130} C_VEL
LIN {X 0,Y 471.931,Z 768.877,A -85,B 0,C 180,E1 23127.814,E2 23127.814} C_VEL
LIN {X 0,Y 472.012,Z 764.166,A -85,B 0,C 180,E1 23125.139,E2 23125.139} C_VEL
LIN {X 0,Y 472.19,Z 758.595,A -85,B 0,C 180,E1 23122.823,E2 23122.823} C_VEL
LIN {X 0,Y 472.571,Z 751.061,A -85,B 0,C 180,E1 23120.378,E2 23120.378} C_VEL
LIN {X 0,Y 473.164,Z 741.988,A -85,B 0,C 180,E1 23118.048,E2 23118.048} C_VEL
LIN {X 0,Y 473.974,Z 731.534,A -85,B 0,C 180,E1 23115.836,E2 23115.836} C_VEL
LIN {X 0,Y 475.073,Z 718.846,A -85,B 0,C 180,E1 23113.619,E2 23113.619} C_VEL
LIN {X 0,Y 476.308,Z 705.305,A -85,B 0,C 180,E1 23111.646,E2 23111.646} C_VEL
LIN {X 0,Y 477.68,Z 690.708,A -85,B 0,C 180,E1 23109.85,E2 23109.85} C_VEL
LIN {X 0,Y 479.175,Z 674.823,A -85,B 0,C 180,E1 23108.197,E2 23108.197} C_VEL
LIN {X 0,Y 480.676,Z 657.917,A -85,B 0,C 180,E1 23106.72,E2 23106.72} C_VEL
LIN {X 0,Y 482.133,Z 640.102,A -85,B 0,C 180,E1 23105.43,E2 23105.43} C_VEL
LIN {X 0,Y 483.485,Z 621.496,A -85,B 0,C 180,E1 23104.326,E2 23104.326} C_VEL
LIN {X 0,Y 484.701,Z 601.855,A -85,B 0,C 180,E1 23103.399,E2 23103.399} C_VEL
LIN {X 0,Y 485.714,Z 581.02,A -85,B 0,C 180,E1 23102.661,E2 23102.661} C_VEL
LIN {X 0,Y 486.43,Z 559.551,A -85,B 0,C 180,E1 23102.142,E2 23102.142} C_VEL
LIN {X 0,Y 490.912,Z 404.564,A -85,B 0,C 180,E1 23099.318,E2 23099.318} C_VEL
LIN {X 0,Y 492.485,Z 322.085,A -85,B 0,C 180,E1 23097.936,E2 23097.936} C_VEL
LIN {X 0,Y 491.823,Z 318.21,A -85,B 0,C 180,E1 23097.778,E2 23097.778} C_VEL
LIN {X 0,Y 493.667,Z 297.611,A -85,B 0,C 180,E1 23095.933,E2 23095.933} C_VEL
LIN {X 0,Y 485.638,Z 279.842,A -85,B 0,C 180,E1 23093.02,E2 23093.02} C_VEL
LIN {X 0,Y 479.085,Z 266.567,A -85,B 0,C 180,E1 23090.62,E2 23090.62} C_VEL
LIN {X 0,Y 476.779,Z 262.069,A -85,B 0,C 180,E1 23089.761,E2 23089.761} C_VEL
LIN {X 0,Y 475.093,Z 258.362,A -85,B 0,C 180,E1 23089.073,E2 23089.073} C_VEL
LIN {X 0,Y 473.244,Z 255.192,A -85,B 0,C 180,E1 23088.412,E2 23088.412} C_VEL
LIN {X 0,Y 472.951,Z 253.824,A -85,B 0,C 180,E1 23088.164,E2 23088.164} C_VEL
LIN {X 0,Y 472.953,Z 253.824,A -85,B 0,C 180,E1 23084.566,E2 23084.566} C_VEL
LIN {X 0,Y 472.949,Z 253.806,A -85,B 0,C 180,E1 23080.788,E2 23080.788} C_VEL
LIN {X 0,Y 472.937,Z 253.807,A -85,B 0,C 180,E1 23077.152,E2 23077.152} C_VEL
LIN {X 0,Y 472.94,Z 253.827,A -85,B 0,C 180,E1 23073.594,E2 23073.594} C_VEL
LIN {X 0,Y 472.981,Z 254.02,A -85,B 0,C 180,E1 23071.578,E2 23071.578} C_VEL
LIN {X 0,Y 480.984,Z 278.993,A -85,B 0,C 180,E1 23068.935,E2 23068.935} C_VEL
LIN {X 0,Y 480.263,Z 321.901,A -85,B 0,C 180,E1 23065.337,E2 23065.337} C_VEL
LIN {X 0,Y 479.383,Z 363.502,A -85,B 0,C 180,E1 23061.851,E2 23061.851} C_VEL
LIN {X 0,Y 478.333,Z 406.243,A -85,B 0,C 180,E1 23058.273,E2 23058.273} C_VEL
LIN {X 0,Y 477.404,Z 447.358,A -85,B 0,C 180,E1 23054.867,E2 23054.867} C_VEL
LIN {X 0,Y 477.568,Z 458.153,A -85,B 0,C 180,E1 23054.675,E2 23054.675} C_VEL
LIN {X 0,Y 476.205,Z 590.516,A -85,B 0,C 180,E1 23052.494,E2 23052.494} C_VEL
LIN {X 0,Y 476.054,Z 606.928,A -85,B 0,C 180,E1 23052.002,E2 23052.002} C_VEL
LIN {X 0,Y 475.753,Z 621.954,A -85,B 0,C 180,E1 23051.333,E2 23051.333} C_VEL
LIN {X 0,Y 475.364,Z 637.219,A -85,B 0,C 180,E1 23050.422,E2 23050.422} C_VEL
LIN {X 0,Y 474.89,Z 651.196,A -85,B 0,C 180,E1 23049.33,E2 23049.33} C_VEL
LIN {X 0,Y 474.412,Z 664.186,A -85,B 0,C 180,E1 23048.057,E2 23048.057} C_VEL
LIN {X 0,Y 473.922,Z 676.399,A -85,B 0,C 180,E1 23046.542,E2 23046.542} C_VEL
LIN {X 0,Y 473.548,Z 685.82,A -85,B 0,C 180,E1 23045.088,E2 23045.088} C_VEL
LIN {X 0,Y 473.208,Z 695.101,A -85,B 0,C 180,E1 23043.271,E2 23043.271} C_VEL
LIN {X 0,Y 473.006,Z 701.731,A -85,B 0,C 180,E1 23041.575,E2 23041.575} C_VEL
LIN {X 0,Y 472.859,Z 707.32,A -85,B 0,C 180,E1 23039.637,E2 23039.637} C_VEL
LIN {X 0,Y 472.796,Z 710.919,A -85,B 0,C 180,E1 23037.698,E2 23037.698} C_VEL
LIN {X 0,Y 472.784,Z 712.781,A -85,B 0,C 180,E1 23035.756,E2 23035.756} C_VEL
LIN {X 0,Y 472.831,Z 712.802,A -85,B 0,C 180,E1 23033.809,E2 23033.809} C_VEL
LIN {X 0,Y 472.909,Z 711.079,A -85,B 0,C 180,E1 23031.857,E2 23031.857} C_VEL
LIN {X 0,Y 473.064,Z 707.423,A -85,B 0,C 180,E1 23029.897,E2 23029.897} C_VEL
LIN {X 0,Y 473.258,Z 702.571,A -85,B 0,C 180,E1 23028.175,E2 23028.175} C_VEL
LIN {X 0,Y 473.533,Z 695.313,A -85,B 0,C 180,E1 23026.321,E2 23026.321} C_VEL
LIN {X 0,Y 473.882,Z 687.029,A -85,B 0,C 180,E1 23024.708,E2 23024.708} C_VEL
LIN {X 0,Y 474.315,Z 676.376,A -85,B 0,C 180,E1 23023.088,E2 23023.088} C_VEL
LIN {X 0,Y 474.746,Z 664.841,A -85,B 0,C 180,E1 23021.712,E2 23021.712} C_VEL
LIN {X 0,Y 475.164,Z 652.267,A -85,B 0,C 180,E1 23020.511,E2 23020.511} C_VEL
LIN {X 0,Y 475.528,Z 637.883,A -85,B 0,C 180,E1 23019.443,E2 23019.443} C_VEL
LIN {X 0,Y 475.79,Z 623.156,A -85,B 0,C 180,E1 23018.611,E2 23018.611} C_VEL
LIN {X 0,Y 475.956,Z 606.401,A -85,B 0,C 180,E1 23017.937,E2 23017.937} C_VEL
LIN {X 0,Y 475.946,Z 589.372,A -85,B 0,C 180,E1 23017.511,E2 23017.511} C_VEL
LIN {X 0,Y 476.919,Z 487.879,A -85,B 0,C 180,E1 23015.843,E2 23015.843} C_VEL
LIN {X 0,Y 477.472,Z 454.785,A -85,B 0,C 180,E1 23015.241,E2 23015.241} C_VEL
LIN {X 0,Y 478.285,Z 449.426,A -85,B 0,C 180,E1 23014.85,E2 23014.85} C_VEL
LIN {X 0,Y 478.86,Z 407.346,A -85,B 0,C 180,E1 23011.528,E2 23011.528} C_VEL
LIN {X 0,Y 479.044,Z 372.768,A -85,B 0,C 180,E1 23008.897,E2 23008.897} C_VEL
LIN {X 0,Y 478.889,Z 331.873,A -85,B 0,C 180,E1 23005.904,E2 23005.904} C_VEL
LIN {X 0,Y 478.83,Z 323.748,A -85,B 0,C 180,E1 23005.319,E2 23005.319} C_VEL
LIN {X 0,Y 480.29,Z 324.532,A -85,B 0,C 180,E1 23005.076,E2 23005.076} C_VEL
LIN {X 0,Y 482.551,Z 324.301,A -85,B 0,C 180,E1 23004.829,E2 23004.829} C_VEL
LIN {X 0,Y 485.103,Z 323.406,A -85,B 0,C 180,E1 23004.608,E2 23004.608} C_VEL
LIN {X 0,Y 488.982,Z 322.837,A -85,B 0,C 180,E1 23004.211,E2 23004.211} C_VEL
LIN {X 0,Y 491.367,Z 322.38,A -85,B 0,C 180,E1 23003.98,E2 23003.98} C_VEL
LIN {X 0,Y 496.846,Z 321.37,A -85,B 0,C 180,E1 23003.458,E2 23003.458} C_VEL
LIN {X 0,Y 495.766,Z 345,A -85,B 0,C 180,E1 23001.678,E2 23001.678} C_VEL
LIN {X 0,Y 496.774,Z 361.979,A -85,B 0,C 180,E1 23000.252,E2 23000.252} C_VEL
LIN {X 0,Y 499.408,Z 376.741,A -85,B 0,C 180,E1 22998.877,E2 22998.877} C_VEL
LIN {X 0,Y 503.584,Z 389.67,A -85,B 0,C 180,E1 22997.541,E2 22997.541} C_VEL
LIN {X 0,Y 509.627,Z 401.564,A -85,B 0,C 180,E1 22996.167,E2 22996.167} C_VEL
LIN {X 0,Y 517.325,Z 411.859,A -85,B 0,C 180,E1 22994.821,E2 22994.821} C_VEL
LIN {X 0,Y 525.955,Z 420.082,A -85,B 0,C 180,E1 22993.59,E2 22993.59} C_VEL
LIN {X 0,Y 536.116,Z 427.002,A -85,B 0,C 180,E1 22992.393,E2 22992.393} C_VEL
LIN {X 0,Y 547.839,Z 432.506,A -85,B 0,C 180,E1 22991.242,E2 22991.242} C_VEL
LIN {X 0,Y 557.824,Z 435.577,A -85,B 0,C 180,E1 22990.379,E2 22990.379} C_VEL
LIN {X 0,Y 558.633,Z 435.912,A -85,B 0,C 180,E1 22990.281,E2 22990.281} C_VEL
LIN {X 0,Y 544.101,Z 457.849,A -85,B 0,C 180,E1 22989.892,E2 22989.892} C_VEL
LIN {X 0,Y 526.145,Z 485.68,A -85,B 0,C 180,E1 22989.259,E2 22989.259} C_VEL
LIN {X 0,Y 517.204,Z 501.788,A -85,B 0,C 180,E1 22988.782,E2 22988.782} C_VEL
LIN {X 0,Y 511.029,Z 515.696,A -85,B 0,C 180,E1 22988.262,E2 22988.262} C_VEL
LIN {X 0,Y 508.364,Z 521.171,A -85,B 0,C 180,E1 22988.068,E2 22988.068} C_VEL
LIN {X 0,Y 501.82,Z 534.898,A -85,B 0,C 180,E1 22987.568,E2 22987.568} C_VEL
LIN {X 0,Y 493.314,Z 558.663,A -85,B 0,C 180,E1 22986.504,E2 22986.504} C_VEL
LIN {X 0,Y 492.644,Z 561.681,A -85,B 0,C 180,E1 22986.392,E2 22986.392} C_VEL
LIN {X 0,Y 491.97,Z 575.09,A -85,B 0,C 180,E1 22986.212,E2 22986.212} C_VEL
LIN {X 0,Y 491.189,Z 607.295,A -85,B 0,C 180,E1 22985.649,E2 22985.649} C_VEL
LIN {X 0,Y 490.062,Z 630.065,A -85,B 0,C 180,E1 22985.053,E2 22985.053} C_VEL
LIN {X 0,Y 488.666,Z 652.617,A -85,B 0,C 180,E1 22984.241,E2 22984.241} C_VEL
LIN {X 0,Y 487.108,Z 674.255,A -85,B 0,C 180,E1 22983.234,E2 22983.234} C_VEL
LIN {X 0,Y 485.474,Z 694.117,A -85,B 0,C 180,E1 22982.098,E2 22982.098} C_VEL
LIN {X 0,Y 483.773,Z 713.515,A -85,B 0,C 180,E1 22980.766,E2 22980.766} C_VEL
LIN {X 0,Y 482,Z 732.026,A -85,B 0,C 180,E1 22979.264,E2 22979.264} C_VEL
LIN {X 0,Y 480.368,Z 748.138,A -85,B 0,C 180,E1 22977.724,E2 22977.724} C_VEL
LIN {X 0,Y 478.469,Z 765.294,A -85,B 0,C 180,E1 22975.755,E2 22975.755} C_VEL
LIN {X 0,Y 476.733,Z 781.459,A -85,B 0,C 180,E1 22973.577,E2 22973.577} C_VEL
LIN {X 0,Y 475.228,Z 796.349,A -85,B 0,C 180,E1 22971.216,E2 22971.216} C_VEL
LIN {X 0,Y 474.027,Z 809.737,A -85,B 0,C 180,E1 22968.7,E2 22968.7} C_VEL
LIN {X 0,Y 473.125,Z 821.41,A -85,B 0,C 180,E1 22966.072,E2 22966.072} C_VEL
LIN {X 0,Y 472.53,Z 830.94,A -85,B 0,C 180,E1 22963.459,E2 22963.459} C_VEL
LIN {X 0,Y 472.174,Z 838.946,A -85,B 0,C 180,E1 22960.721,E2 22960.721} C_VEL
LIN {X 0,Y 472.003,Z 844.915,A -85,B 0,C 180,E1 22958.037,E2 22958.037} C_VEL
LIN {X 0,Y 471.932,Z 848.979,A -85,B 0,C 180,E1 22955.471,E2 22955.471} C_VEL
LIN {X 0,Y 471.911,Z 851.573,A -85,B 0,C 180,E1 22952.793,E2 22952.793} C_VEL
LIN {X 0,Y 471.909,Z 852.489,A -85,B 0,C 180,E1 22950.121,E2 22950.121} C_VEL
LIN {X 0,Y 471.909,Z 851.78,A -85,B 0,C 180,E1 22947.571,E2 22947.571} C_VEL
LIN {X 0,Y 471.927,Z 849.59,A -85,B 0,C 180,E1 22945.017,E2 22945.017} C_VEL
LIN {X 0,Y 471.981,Z 845.598,A -85,B 0,C 180,E1 22942.33,E2 22942.33} C_VEL
LIN {X 0,Y 472.144,Z 839.811,A -85,B 0,C 180,E1 22939.63,E2 22939.63} C_VEL
LIN {X 0,Y 472.45,Z 832.526,A -85,B 0,C 180,E1 22937.036,E2 22937.036} C_VEL
LIN {X 0,Y 472.952,Z 823.857,A -85,B 0,C 180,E1 22934.551,E2 22934.551} C_VEL
LIN {X 0,Y 473.77,Z 812.719,A -85,B 0,C 180,E1 22931.926,E2 22931.926} C_VEL
LIN {X 0,Y 474.89,Z 799.921,A -85,B 0,C 180,E1 22929.414,E2 22929.414} C_VEL
LIN {X 0,Y 476.314,Z 785.455,A -85,B 0,C 180,E1 22927.018,E2 22927.018} C_VEL
LIN {X 0,Y 478.042,Z 769.236,A -85,B 0,C 180,E1 22924.743,E2 22924.743} C_VEL
LIN {X 0,Y 479.991,Z 751.684,A -85,B 0,C 180,E1 22922.657,E2 22922.657} C_VEL
LIN {X 0,Y 481.56,Z 736.58,A -85,B 0,C 180,E1 22921.142,E2 22921.142} C_VEL
LIN {X 0,Y 483.486,Z 716.585,A -85,B 0,C 180,E1 22919.468,E2 22919.468} C_VEL
LIN {X 0,Y 485.296,Z 696.102,A -85,B 0,C 180,E1 22918.028,E2 22918.028} C_VEL
LIN {X 0,Y 487.027,Z 674.992,A -85,B 0,C 180,E1 22916.812,E2 22916.812} C_VEL
LIN {X 0,Y 488.633,Z 652.34,A -85,B 0,C 180,E1 22915.759,E2 22915.759} C_VEL
LIN {X 0,Y 490.052,Z 629.455,A -85,B 0,C 180,E1 22914.939,E2 22914.939} C_VEL
LIN {X 0,Y 491.142,Z 607.009,A -85,B 0,C 180,E1 22914.356,E2 22914.356} C_VEL
LIN {X 0,Y 491.966,Z 572.783,A -85,B 0,C 180,E1 22913.759,E2 22913.759} C_VEL
LIN {X 0,Y 492.865,Z 561.318,A -85,B 0,C 180,E1 22913.62,E2 22913.62} C_VEL
LIN {X 0,Y 497.31,Z 550.578,A -85,B 0,C 180,E1 22913.047,E2 22913.047} C_VEL
LIN {X 0,Y 504.009,Z 536.204,A -85,B 0,C 180,E1 22912.337,E2 22912.337} C_VEL
LIN {X 0,Y 512.006,Z 523.304,A -85,B 0,C 180,E1 22911.824,E2 22911.824} C_VEL
LIN {X 0,Y 521.016,Z 507.643,A -85,B 0,C 180,E1 22911.181,E2 22911.181} C_VEL
LIN {X 0,Y 531.357,Z 493.06,A -85,B 0,C 180,E1 22910.713,E2 22910.713} C_VEL
LIN {X 0,Y 550.781,Z 468.501,A -85,B 0,C 180,E1 22910.084,E2 22910.084} C_VEL
LIN {X 0,Y 538.036,Z 463.778,A -85,B 0,C 180,E1 22908.98,E2 22908.98} C_VEL
LIN {X 0,Y 526.571,Z 457.421,A -85,B 0,C 180,E1 22907.777,E2 22907.777} C_VEL
LIN {X 0,Y 516.79,Z 449.686,A -85,B 0,C 180,E1 22906.513,E2 22906.513} C_VEL
LIN {X 0,Y 508.707,Z 440.679,A -85,B 0,C 180,E1 22905.197,E2 22905.197} C_VEL
LIN {X 0,Y 502.747,Z 431.351,A -85,B 0,C 180,E1 22903.95,E2 22903.95} C_VEL
LIN {X 0,Y 497.915,Z 420.216,A -85,B 0,C 180,E1 22902.588,E2 22902.588} C_VEL
LIN {X 0,Y 494.478,Z 406.66,A -85,B 0,C 180,E1 22901.084,E2 22901.084} C_VEL
LIN {X 0,Y 492.833,Z 391.593,A -85,B 0,C 180,E1 22899.561,E2 22899.561} C_VEL
LIN {X 0,Y 493.095,Z 373.531,A -85,B 0,C 180,E1 22897.908,E2 22897.908} C_VEL
LIN {X 0,Y 497.064,Z 330.154,A -85,B 0,C 180,E1 22894.14,E2 22894.14} C_VEL
LIN {X 0,Y 499.306,Z 307.533,A -85,B 0,C 180,E1 22892.106,E2 22892.106} C_VEL
LIN {X 0,Y 492.201,Z 291.923,A -85,B 0,C 180,E1 22889.445,E2 22889.445} C_VEL
LIN {X 0,Y 490.9,Z 289.337,A -85,B 0,C 180,E1 22888.963,E2 22888.963} C_VEL
LIN {X 0,Y 488.128,Z 290.132,A -85,B 0,C 180,E1 22888.64,E2 22888.64} C_VEL
LIN {X 0,Y 484.35,Z 291.392,A -85,B 0,C 180,E1 22888.211,E2 22888.211} C_VEL
LIN {X 0,Y 482.936,Z 291.724,A -85,B 0,C 180,E1 22888.032,E2 22888.032} C_VEL
LIN {X 0,Y 480.214,Z 293.014,A -85,B 0,C 180,E1 22887.76,E2 22887.76} C_VEL
LIN {X 0,Y 478.516,Z 293.104,A -85,B 0,C 180,E1 22887.502,E2 22887.502} C_VEL
LIN {X 0,Y 477.825,Z 292.82,A -85,B 0,C 180,E1 22887.342,E2 22887.342} C_VEL
LIN {X 0,Y 478.369,Z 336.142,A -85,B 0,C 180,E1 22884.446,E2 22884.446} C_VEL
LIN {X 0,Y 478.354,Z 375.345,A -85,B 0,C 180,E1 22881.713,E2 22881.713} C_VEL
LIN {X 0,Y 478.063,Z 417.274,A -85,B 0,C 180,E1 22878.708,E2 22878.708} C_VEL
LIN {X 0,Y 477.45,Z 461.025,A -85,B 0,C 180,E1 22875.486,E2 22875.486} C_VEL
LIN {X 0,Y 476.756,Z 497.888,A -85,B 0,C 180,E1 22872.721,E2 22872.721} C_VEL
LIN {X 0,Y 476.076,Z 502.738,A -85,B 0,C 180,E1 22872.416,E2 22872.416} C_VEL
LIN {X 0,Y 475.134,Z 615.968,A -85,B 0,C 180,E1 22870.518,E2 22870.518} C_VEL
LIN {X 0,Y 475.095,Z 631.061,A -85,B 0,C 180,E1 22870.029,E2 22870.029} C_VEL
LIN {X 0,Y 474.962,Z 644.219,A -85,B 0,C 180,E1 22869.389,E2 22869.389} C_VEL
LIN {X 0,Y 474.711,Z 657.153,A -85,B 0,C 180,E1 22868.539,E2 22868.539} C_VEL
LIN {X 0,Y 474.408,Z 669.707,A -85,B 0,C 180,E1 22867.447,E2 22867.447} C_VEL
LIN {X 0,Y 474.056,Z 680.944,A -85,B 0,C 180,E1 22866.175,E2 22866.175} C_VEL
LIN {X 0,Y 473.74,Z 690.113,A -85,B 0,C 180,E1 22864.842,E2 22864.842} C_VEL
LIN {X 0,Y 473.452,Z 697.935,A -85,B 0,C 180,E1 22863.39,E2 22863.39} C_VEL
LIN {X 0,Y 473.193,Z 704.735,A -85,B 0,C 180,E1 22861.695,E2 22861.695} C_VEL
LIN {X 0,Y 473.01,Z 709.739,A -85,B 0,C 180,E1 22859.878,E2 22859.878} C_VEL
LIN {X 0,Y 472.892,Z 712.673,A -85,B 0,C 180,E1 22858.061,E2 22858.061} C_VEL
LIN {X 0,Y 472.834,Z 713.698,A -85,B 0,C 180,E1 22856.362,E2 22856.362} C_VEL
LIN {X 0,Y 472.815,Z 713.007,A -85,B 0,C 180,E1 22854.539,E2 22854.539} C_VEL
LIN {X 0,Y 472.853,Z 710.42,A -85,B 0,C 180,E1 22852.711,E2 22852.711} C_VEL
LIN {X 0,Y 472.956,Z 705.735,A -85,B 0,C 180,E1 22850.85,E2 22850.85} C_VEL
LIN {X 0,Y 473.132,Z 699.45,A -85,B 0,C 180,E1 22849.159,E2 22849.159} C_VEL
LIN {X 0,Y 473.365,Z 692.139,A -85,B 0,C 180,E1 22847.682,E2 22847.682} C_VEL
LIN {X 0,Y 473.684,Z 682.684,A -85,B 0,C 180,E1 22846.2,E2 22846.2} C_VEL
LIN {X 0,Y 474.047,Z 671.476,A -85,B 0,C 180,E1 22844.838,E2 22844.838} C_VEL
LIN {X 0,Y 474.405,Z 658.909,A -85,B 0,C 180,E1 22843.658,E2 22843.658} C_VEL
LIN {X 0,Y 474.73,Z 645.906,A -85,B 0,C 180,E1 22842.724,E2 22842.724} C_VEL
LIN {X 0,Y 474.961,Z 632.581,A -85,B 0,C 180,E1 22842.005,E2 22842.005} C_VEL
LIN {X 0,Y 475.116,Z 617.619,A -85,B 0,C 180,E1 22841.443,E2 22841.443} C_VEL
LIN {X 0,Y 475.148,Z 600.954,A -85,B 0,C 180,E1 22841.087,E2 22841.087} C_VEL
LIN {X 0,Y 476.111,Z 496.57,A -85,B 0,C 180,E1 22839.405,E2 22839.405} C_VEL
LIN {X 0,Y 477.115,Z 451.092,A -85,B 0,C 180,E1 22835.88,E2 22835.88} C_VEL
LIN {X 0,Y 478.213,Z 404.687,A -85,B 0,C 180,E1 22832.276,E2 22832.276} C_VEL
LIN {X 0,Y 479.181,Z 359.439,A -85,B 0,C 180,E1 22828.762,E2 22828.762} C_VEL
LIN {X 0,Y 479.99,Z 316.435,A -85,B 0,C 180,E1 22825.414,E2 22825.414} C_VEL
LIN {X 0,Y 480.668,Z 277.826,A -85,B 0,C 180,E1 22822.424,E2 22822.424} C_VEL
LIN {X 0,Y 478.01,Z 269.419,A -85,B 0,C 180,E1 22821.613,E2 22821.613} C_VEL
LIN {X 0,Y 476.873,Z 266.954,A -85,B 0,C 180,E1 22821.233,E2 22821.233} C_VEL
LIN {X 0,Y 475.375,Z 265.526,A -85,B 0,C 180,E1 22820.644,E2 22820.644} C_VEL
LIN {X 0,Y 473.828,Z 265.617,A -85,B 0,C 180,E1 22819.873,E2 22819.873} C_VEL
LIN {X 0,Y 472.634,Z 267.749,A -85,B 0,C 180,E1 22818.843,E2 22818.843} C_VEL
LIN {X 0,Y 472.871,Z 270.794,A -85,B 0,C 180,E1 22817.904,E2 22817.904} C_VEL
LIN {X 0,Y 473.424,Z 272.003,A -85,B 0,C 180,E1 22817.581,E2 22817.581} C_VEL
LIN {X 0,Y 478.324,Z 281.998,A -85,B 0,C 180,E1 22815.215,E2 22815.215} C_VEL
LIN {X 0,Y 483.947,Z 295.005,A -85,B 0,C 180,E1 22812.474,E2 22812.474} C_VEL
LIN {X 0,Y 487.477,Z 303.894,A -85,B 0,C 180,E1 22810.761,E2 22810.761} C_VEL
LIN {X 0,Y 485.26,Z 323.333,A -85,B 0,C 180,E1 22808.655,E2 22808.655} C_VEL
LIN {X 0,Y 486.342,Z 328.539,A -85,B 0,C 180,E1 22808.455,E2 22808.455} C_VEL
LIN {X 0,Y 484.144,Z 418.875,A -85,B 0,C 180,E1 22806.917,E2 22806.917} C_VEL
LIN {X 0,Y 479.877,Z 546.405,A -85,B 0,C 180,E1 22804.491,E2 22804.491} C_VEL
LIN {X 0,Y 478.887,Z 575.514,A -85,B 0,C 180,E1 22803.857,E2 22803.857} C_VEL
LIN {X 0,Y 477.985,Z 594.899,A -85,B 0,C 180,E1 22803.234,E2 22803.234} C_VEL
LIN {X 0,Y 476.733,Z 615.612,A -85,B 0,C 180,E1 22802.332,E2 22802.332} C_VEL
LIN {X 0,Y 475.305,Z 635.221,A -85,B 0,C 180,E1 22801.235,E2 22801.235} C_VEL
LIN {X 0,Y 473.731,Z 654.078,A -85,B 0,C 180,E1 22799.924,E2 22799.924} C_VEL
LIN {X 0,Y 472.063,Z 672.173,A -85,B 0,C 180,E1 22798.393,E2 22798.393} C_VEL
LIN {X 0,Y 470.396,Z 689.264,A -85,B 0,C 180,E1 22796.647,E2 22796.647} C_VEL
LIN {X 0,Y 468.871,Z 704.571,A -85,B 0,C 180,E1 22794.774,E2 22794.774} C_VEL
LIN {X 0,Y 467.507,Z 718.271,A -85,B 0,C 180,E1 22792.775,E2 22792.775} C_VEL
LIN {X 0,Y 466.388,Z 730.156,A -85,B 0,C 180,E1 22790.716,E2 22790.716} C_VEL
LIN {X 0,Y 465.485,Z 740.719,A -85,B 0,C 180,E1 22788.536,E2 22788.536} C_VEL
LIN {X 0,Y 464.814,Z 749.924,A -85,B 0,C 180,E1 22786.239,E2 22786.239} C_VEL
LIN {X 0,Y 464.358,Z 757.783,A -85,B 0,C 180,E1 22783.807,E2 22783.807} C_VEL
LIN {X 0,Y 464.084,Z 764.253,A -85,B 0,C 180,E1 22781.181,E2 22781.181} C_VEL
LIN {X 0,Y 463.971,Z 768.469,A -85,B 0,C 180,E1 22778.801,E2 22778.801} C_VEL
LIN {X 0,Y 463.925,Z 771.373,A -85,B 0,C 180,E1 22776.311,E2 22776.311} C_VEL
LIN {X 0,Y 463.911,Z 772.643,A -85,B 0,C 180,E1 22773.707,E2 22773.707} C_VEL
LIN {X 0,Y 463.91,Z 772.421,A -85,B 0,C 180,E1 22771.359,E2 22771.359} C_VEL
LIN {X 0,Y 463.929,Z 770.58,A -85,B 0,C 180,E1 22768.765,E2 22768.765} C_VEL
LIN {X 0,Y 463.987,Z 767.383,A -85,B 0,C 180,E1 22766.417,E2 22766.417} C_VEL
LIN {X 0,Y 464.147,Z 762.505,A -85,B 0,C 180,E1 22763.941,E2 22763.941} C_VEL
LIN {X 0,Y 464.453,Z 755.829,A -85,B 0,C 180,E1 22761.458,E2 22761.458} C_VEL
LIN {X 0,Y 464.966,Z 747.79,A -85,B 0,C 180,E1 22759.092,E2 22759.092} C_VEL
LIN {X 0,Y 465.735,Z 737.785,A -85,B 0,C 180,E1 22756.72,E2 22756.72} C_VEL
LIN {X 0,Y 466.753,Z 726.227,A -85,B 0,C 180,E1 22754.468,E2 22754.468} C_VEL
LIN {X 0,Y 468.014,Z 713.049,A -85,B 0,C 180,E1 22752.333,E2 22752.333} C_VEL
LIN {X 0,Y 469.424,Z 698.826,A -85,B 0,C 180,E1 22750.399,E2 22750.399} C_VEL
LIN {X 0,Y 470.887,Z 684.102,A -85,B 0,C 180,E1 22748.71,E2 22748.71} C_VEL
LIN {X 0,Y 472.442,Z 668.03,A -85,B 0,C 180,E1 22747.148,E2 22747.148} C_VEL
LIN {X 0,Y 473.956,Z 651.259,A -85,B 0,C 180,E1 22745.775,E2 22745.775} C_VEL
LIN {X 0,Y 475.423,Z 633.977,A -85,B 0,C 180,E1 22744.594,E2 22744.594} C_VEL
LIN {X 0,Y 476.853,Z 614.394,A -85,B 0,C 180,E1 22743.51,E2 22743.51} C_VEL
LIN {X 0,Y 478.05,Z 594.204,A -85,B 0,C 180,E1 22742.642,E2 22742.642} C_VEL
LIN {X 0,Y 478.993,Z 573.375,A -85,B 0,C 180,E1 22741.987,E2 22741.987} C_VEL
LIN {X 0,Y 480.413,Z 530.179,A -85,B 0,C 180,E1 22741.103,E2 22741.103} C_VEL
LIN {X 0,Y 484.301,Z 409.736,A -85,B 0,C 180,E1 22738.853,E2 22738.853} C_VEL
LIN {X 0,Y 486.085,Z 323.516,A -85,B 0,C 180,E1 22737.388,E2 22737.388} C_VEL
LIN {X 0,Y 485.541,Z 320.732,A -85,B 0,C 180,E1 22737.278,E2 22737.278} C_VEL
LIN {X 0,Y 487.327,Z 301.738,A -85,B 0,C 180,E1 22735.568,E2 22735.568} C_VEL
LIN {X 0,Y 479.747,Z 284.887,A -85,B 0,C 180,E1 22732.764,E2 22732.764} C_VEL
LIN {X 0,Y 473.343,Z 271.786,A -85,B 0,C 180,E1 22730.362,E2 22730.362} C_VEL
LIN {X 0,Y 469.267,Z 263.633,A -85,B 0,C 180,E1 22728.776,E2 22728.776} C_VEL
LIN {X 0,Y 467.249,Z 259.447,A -85,B 0,C 180,E1 22727.949,E2 22727.949} C_VEL
LIN {X 0,Y 465.303,Z 256.205,A -85,B 0,C 180,E1 22727.232,E2 22727.232} C_VEL
LIN {X 0,Y 465.011,Z 254.812,A -85,B 0,C 180,E1 22726.976,E2 22726.976} C_VEL
LIN {X 0,Y 465.003,Z 254.812,A -85,B 0,C 180,E1 22723.203,E2 22723.203} C_VEL
LIN {X 0,Y 464.997,Z 254.808,A -85,B 0,C 180,E1 22719.53,E2 22719.53} C_VEL
LIN {X 0,Y 465.008,Z 254.799,A -85,B 0,C 180,E1 22715.945,E2 22715.945} C_VEL
LIN {X 0,Y 465.017,Z 254.813,A -85,B 0,C 180,E1 22712.225,E2 22712.225} C_VEL
LIN {X 0,Y 465.044,Z 254.996,A -85,B 0,C 180,E1 22712.025,E2 22712.025} C_VEL
LIN {X 0,Y 473.374,Z 280.705,A -85,B 0,C 180,E1 22709.268,E2 22709.268} C_VEL
LIN {X 0,Y 473.382,Z 292.704,A -85,B 0,C 180,E1 22708.238,E2 22708.238} C_VEL
LIN {X 0,Y 472.63,Z 333.103,A -85,B 0,C 180,E1 22704.829,E2 22704.829} C_VEL
LIN {X 0,Y 471.607,Z 375.846,A -85,B 0,C 180,E1 22701.222,E2 22701.222} C_VEL
LIN {X 0,Y 470.541,Z 417.862,A -85,B 0,C 180,E1 22697.69,E2 22697.69} C_VEL
LIN {X 0,Y 469.843,Z 448.459,A -85,B 0,C 180,E1 22695.155,E2 22695.155} C_VEL
LIN {X 0,Y 469.762,Z 473.733,A -85,B 0,C 180,E1 22694.714,E2 22694.714} C_VEL
LIN {X 0,Y 468.476,Z 591.707,A -85,B 0,C 180,E1 22692.722,E2 22692.722} C_VEL
LIN {X 0,Y 468.315,Z 608.589,A -85,B 0,C 180,E1 22692.203,E2 22692.203} C_VEL
LIN {X 0,Y 467.973,Z 624.635,A -85,B 0,C 180,E1 22691.462,E2 22691.462} C_VEL
LIN {X 0,Y 467.561,Z 639.539,A -85,B 0,C 180,E1 22690.536,E2 22690.536} C_VEL
LIN {X 0,Y 467.058,Z 654.039,A -85,B 0,C 180,E1 22689.364,E2 22689.364} C_VEL
LIN {X 0,Y 466.556,Z 666.702,A -85,B 0,C 180,E1 22688.068,E2 22688.068} C_VEL
LIN {X 0,Y 466.093,Z 677.852,A -85,B 0,C 180,E1 22686.653,E2 22686.653} C_VEL
LIN {X 0,Y 465.666,Z 687.947,A -85,B 0,C 180,E1 22685.051,E2 22685.051} C_VEL
LIN {X 0,Y 465.345,Z 696.562,A -85,B 0,C 180,E1 22683.326,E2 22683.326} C_VEL
LIN {X 0,Y 465.115,Z 703.584,A -85,B 0,C 180,E1 22681.479,E2 22681.479} C_VEL
LIN {X 0,Y 464.976,Z 708.767,A -85,B 0,C 180,E1 22679.631,E2 22679.631} C_VEL
LIN {X 0,Y 464.909,Z 712.346,A -85,B 0,C 180,E1 22677.659,E2 22677.659} C_VEL
LIN {X 0,Y 464.901,Z 714.17,A -85,B 0,C 180,E1 22675.683,E2 22675.683} C_VEL
LIN {X 0,Y 464.957,Z 714.158,A -85,B 0,C 180,E1 22673.704,E2 22673.704} C_VEL
LIN {X 0,Y 465.044,Z 712.546,A -85,B 0,C 180,E1 22671.843,E2 22671.843} C_VEL
LIN {X 0,Y 465.215,Z 708.926,A -85,B 0,C 180,E1 22669.85,E2 22669.85} C_VEL
LIN {X 0,Y 465.428,Z 704.094,A -85,B 0,C 180,E1 22668.099,E2 22668.099} C_VEL
LIN {X 0,Y 465.726,Z 696.832,A -85,B 0,C 180,E1 22666.214,E2 22666.214} C_VEL
LIN {X 0,Y 466.102,Z 688.54,A -85,B 0,C 180,E1 22664.574,E2 22664.574} C_VEL
LIN {X 0,Y 466.568,Z 677.882,A -85,B 0,C 180,E1 22662.927,E2 22662.927} C_VEL
LIN {X 0,Y 467.028,Z 666.241,A -85,B 0,C 180,E1 22661.518,E2 22661.518} C_VEL
LIN {X 0,Y 467.46,Z 653.763,A -85,B 0,C 180,E1 22660.314,E2 22660.314} C_VEL
LIN {X 0,Y 467.814,Z 640.148,A -85,B 0,C 180,E1 22659.285,E2 22659.285} C_VEL
LIN {X 0,Y 468.087,Z 625.76,A -85,B 0,C 180,E1 22658.445,E2 22658.445} C_VEL
LIN {X 0,Y 468.257,Z 609.198,A -85,B 0,C 180,E1 22657.753,E2 22657.753} C_VEL
LIN {X 0,Y 468.257,Z 593.003,A -85,B 0,C 180,E1 22657.317,E2 22657.317} C_VEL
LIN {X 0,Y 469.329,Z 489.269,A -85,B 0,C 180,E1 22655.553,E2 22655.553} C_VEL
LIN {X 0,Y 469.911,Z 456.896,A -85,B 0,C 180,E1 22654.949,E2 22654.949} C_VEL
LIN {X 0,Y 470.912,Z 450.229,A -85,B 0,C 180,E1 22654.468,E2 22654.468} C_VEL
LIN {X 0,Y 471.483,Z 411.479,A -85,B 0,C 180,E1 22651.398,E2 22651.398} C_VEL
LIN {X 0,Y 471.73,Z 375.24,A -85,B 0,C 180,E1 22648.622,E2 22648.622} C_VEL
LIN {X 0,Y 471.621,Z 336.552,A -85,B 0,C 180,E1 22645.774,E2 22645.774} C_VEL
LIN {X 0,Y 471.631,Z 332.189,A -85,B 0,C 180,E1 22645.452,E2 22645.452} C_VEL
LIN {X 0,Y 473.099,Z 332.944,A -85,B 0,C 180,E1 22645.207,E2 22645.207} C_VEL
LIN {X 0,Y 475.382,Z 332.652,A -85,B 0,C 180,E1 22644.957,E2 22644.957} C_VEL
LIN {X 0,Y 477.613,Z 331.654,A -85,B 0,C 180,E1 22644.779,E2 22644.779} C_VEL
LIN {X 0,Y 481.847,Z 331.085,A -85,B 0,C 180,E1 22644.332,E2 22644.332} C_VEL
LIN {X 0,Y 484.295,Z 330.473,A -85,B 0,C 180,E1 22644.103,E2 22644.103} C_VEL
LIN {X 0,Y 490.084,Z 329.393,A -85,B 0,C 180,E1 22643.543,E2 22643.543} C_VEL
LIN {X 0,Y 489.351,Z 350.88,A -85,B 0,C 180,E1 22641.874,E2 22641.874} C_VEL
LIN {X 0,Y 490.636,Z 368.226,A -85,B 0,C 180,E1 22640.368,E2 22640.368} C_VEL
LIN {X 0,Y 493.492,Z 382.771,A -85,B 0,C 180,E1 22638.971,E2 22638.971} C_VEL
LIN {X 0,Y 497.987,Z 395.888,A -85,B 0,C 180,E1 22637.576,E2 22637.576} C_VEL
LIN {X 0,Y 504.127,Z 407.536,A -85,B 0,C 180,E1 22636.197,E2 22636.197} C_VEL
LIN {X 0,Y 511.898,Z 417.751,A -85,B 0,C 180,E1 22634.84,E2 22634.84} C_VEL
LIN {X 0,Y 520.587,Z 426.022,A -85,B 0,C 180,E1 22633.592,E2 22633.592} C_VEL
LIN {X 0,Y 530.648,Z 432.982,A -85,B 0,C 180,E1 22632.387,E2 22632.387} C_VEL
LIN {X 0,Y 542.313,Z 438.67,A -85,B 0,C 180,E1 22631.217,E2 22631.217} C_VEL
LIN {X 0,Y 548.098,Z 440.912,A -85,B 0,C 180,E1 22630.696,E2 22630.696} C_VEL
LIN {X 0,Y 522.943,Z 478.922,A -85,B 0,C 180,E1 22629.902,E2 22629.902} C_VEL
LIN {X 0,Y 512.277,Z 497.409,A -85,B 0,C 180,E1 22629.385,E2 22629.385} C_VEL
LIN {X 0,Y 505.307,Z 512.307,A -85,B 0,C 180,E1 22628.848,E2 22628.848} C_VEL
LIN {X 0,Y 502.858,Z 517.874,A -85,B 0,C 180,E1 22628.634,E2 22628.634} C_VEL
LIN {X 0,Y 495.711,Z 532.456,A -85,B 0,C 180,E1 22628.113,E2 22628.113} C_VEL
LIN {X 0,Y 486.371,Z 558.072,A -85,B 0,C 180,E1 22626.964,E2 22626.964} C_VEL
LIN {X 0,Y 485.341,Z 573.039,A -85,B 0,C 180,E1 22626.767,E2 22626.767} C_VEL
LIN {X 0,Y 484.505,Z 605.451,A -85,B 0,C 180,E1 22626.194,E2 22626.194} C_VEL
LIN {X 0,Y 483.248,Z 629.011,A -85,B 0,C 180,E1 22625.574,E2 22625.574} C_VEL
LIN {X 0,Y 481.739,Z 651.486,A -85,B 0,C 180,E1 22624.754,E2 22624.754} C_VEL
LIN {X 0,Y 480.134,Z 672.378,A -85,B 0,C 180,E1 22623.781,E2 22623.781} C_VEL
LIN {X 0,Y 478.31,Z 693.482,A -85,B 0,C 180,E1 22622.567,E2 22622.567} C_VEL
LIN {X 0,Y 476.325,Z 714.592,A -85,B 0,C 180,E1 22621.09,E2 22621.09} C_VEL
LIN {X 0,Y 474.432,Z 733.084,A -85,B 0,C 180,E1 22619.548,E2 22619.548} C_VEL
LIN {X 0,Y 472.514,Z 751.508,A -85,B 0,C 180,E1 22617.745,E2 22617.745} C_VEL
LIN {X 0,Y 470.588,Z 769.214,A -85,B 0,C 180,E1 22615.686,E2 22615.686} C_VEL
LIN {X 0,Y 468.809,Z 784.661,A -85,B 0,C 180,E1 22613.497,E2 22613.497} C_VEL
LIN {X 0,Y 467.317,Z 798.495,A -85,B 0,C 180,E1 22611.198,E2 22611.198} C_VEL
LIN {X 0,Y 466.123,Z 810.93,A -85,B 0,C 180,E1 22608.769,E2 22608.769} C_VEL
LIN {X 0,Y 465.212,Z 821.899,A -85,B 0,C 180,E1 22606.225,E2 22606.225} C_VEL
LIN {X 0,Y 464.574,Z 831.351,A -85,B 0,C 180,E1 22603.568,E2 22603.568} C_VEL
LIN {X 0,Y 464.19,Z 839.207,A -85,B 0,C 180,E1 22600.801,E2 22600.801} C_VEL
LIN {X 0,Y 464.007,Z 845.153,A -85,B 0,C 180,E1 22598.052,E2 22598.052} C_VEL
LIN {X 0,Y 463.932,Z 849.132,A -85,B 0,C 180,E1 22595.441,E2 22595.441} C_VEL
LIN {X 0,Y 463.912,Z 851.574,A -85,B 0,C 180,E1 22592.841,E2 22592.841} C_VEL
LIN {X 0,Y 463.909,Z 852.489,A -85,B 0,C 180,E1 22590.123,E2 22590.123} C_VEL
LIN {X 0,Y 463.909,Z 851.782,A -85,B 0,C 180,E1 22587.529,E2 22587.529} C_VEL
LIN {X 0,Y 463.928,Z 849.591,A -85,B 0,C 180,E1 22584.93,E2 22584.93} C_VEL
LIN {X 0,Y 463.992,Z 845.599,A -85,B 0,C 180,E1 22582.197,E2 22582.197} C_VEL
LIN {X 0,Y 464.17,Z 839.812,A -85,B 0,C 180,E1 22579.45,E2 22579.45} C_VEL
LIN {X 0,Y 464.506,Z 832.525,A -85,B 0,C 180,E1 22576.811,E2 22576.811} C_VEL
LIN {X 0,Y 465.06,Z 823.856,A -85,B 0,C 180,E1 22574.282,E2 22574.282} C_VEL
LIN {X 0,Y 465.958,Z 812.718,A -85,B 0,C 180,E1 22571.613,E2 22571.613} C_VEL
LIN {X 0,Y 467.176,Z 799.924,A -85,B 0,C 180,E1 22569.058,E2 22569.058} C_VEL
LIN {X 0,Y 468.723,Z 785.457,A -85,B 0,C 180,E1 22566.624,E2 22566.624} C_VEL
LIN {X 0,Y 470.533,Z 769.72,A -85,B 0,C 180,E1 22564.378,E2 22564.378} C_VEL
LIN {X 0,Y 472.383,Z 752.684,A -85,B 0,C 180,E1 22562.384,E2 22562.384} C_VEL
LIN {X 0,Y 474.279,Z 734.486,A -85,B 0,C 180,E1 22560.58,E2 22560.58} C_VEL
LIN {X 0,Y 476.283,Z 714.657,A -85,B 0,C 180,E1 22558.927,E2 22558.927} C_VEL
LIN {X 0,Y 478.203,Z 694.379,A -85,B 0,C 180,E1 22557.496,E2 22557.496} C_VEL
LIN {X 0,Y 480.019,Z 673.386,A -85,B 0,C 180,E1 22556.281,E2 22556.281} C_VEL
LIN {X 0,Y 481.734,Z 650.834,A -85,B 0,C 180,E1 22555.232,E2 22555.232} C_VEL
LIN {X 0,Y 483.262,Z 627.482,A -85,B 0,C 180,E1 22554.395,E2 22554.395} C_VEL
LIN {X 0,Y 484.448,Z 604.882,A -85,B 0,C 180,E1 22553.809,E2 22553.809} C_VEL
LIN {X 0,Y 485.35,Z 569.956,A -85,B 0,C 180,E1 22553.195,E2 22553.195} C_VEL
LIN {X 0,Y 486.595,Z 558.507,A -85,B 0,C 180,E1 22553.056,E2 22553.056} C_VEL
LIN {X 0,Y 496.303,Z 536.833,A -85,B 0,C 180,E1 22551.941,E2 22551.941} C_VEL
LIN {X 0,Y 504.121,Z 523.659,A -85,B 0,C 180,E1 22551.393,E2 22551.393} C_VEL
LIN {X 0,Y 507.379,Z 518.512,A -85,B 0,C 180,E1 22551.195,E2 22551.195} C_VEL
LIN {X 0,Y 514.477,Z 506.157,A -85,B 0,C 180,E1 22550.686,E2 22550.686} C_VEL
LIN {X 0,Y 524.912,Z 491.329,A -85,B 0,C 180,E1 22550.206,E2 22550.206} C_VEL
LIN {X 0,Y 539.546,Z 472.648,A -85,B 0,C 180,E1 22549.717,E2 22549.717} C_VEL
LIN {X 0,Y 527.834,Z 467.29,A -85,B 0,C 180,E1 22548.601,E2 22548.601} C_VEL
LIN {X 0,Y 517.45,Z 460.617,A -85,B 0,C 180,E1 22547.408,E2 22547.408} C_VEL
LIN {X 0,Y 508.025,Z 452.244,A -85,B 0,C 180,E1 22546.082,E2 22546.082} C_VEL
LIN {X 0,Y 500.338,Z 442.677,A -85,B 0,C 180,E1 22544.702,E2 22544.702} C_VEL
LIN {X 0,Y 494.22,Z 431.642,A -85,B 0,C 180,E1 22543.254,E2 22543.254} C_VEL
LIN {X 0,Y 489.849,Z 419.439,A -85,B 0,C 180,E1 22541.792,E2 22541.792} C_VEL
LIN {X 0,Y 487.047,Z 404.909,A -85,B 0,C 180,E1 22540.21,E2 22540.21} C_VEL
LIN {X 0,Y 486.102,Z 388.571,A -85,B 0,C 180,E1 22538.59,E2 22538.59} C_VEL
LIN {X 0,Y 487.466,Z 366.036,A -85,B 0,C 180,E1 22536.573,E2 22536.573} C_VEL
LIN {X 0,Y 491.522,Z 326.295,A -85,B 0,C 180,E1 22533.06,E2 22533.06} C_VEL
LIN {X 0,Y 493.111,Z 311.839,A -85,B 0,C 180,E1 22531.747,E2 22531.747} C_VEL
LIN {X 0,Y 486.323,Z 296.777,A -85,B 0,C 180,E1 22529.135,E2 22529.135} C_VEL
LIN {X 0,Y 481.167,Z 298.439,A -85,B 0,C 180,E1 22528.55,E2 22528.55} C_VEL
LIN {X 0,Y 477.268,Z 299.874,A -85,B 0,C 180,E1 22528.117,E2 22528.117} C_VEL
LIN {X 0,Y 475.978,Z 300.031,A -85,B 0,C 180,E1 22527.933,E2 22527.933} C_VEL
LIN {X 0,Y 472.782,Z 301.569,A -85,B 0,C 180,E1 22527.609,E2 22527.609} C_VEL
LIN {X 0,Y 470.677,Z 301.375,A -85,B 0,C 180,E1 22527.244,E2 22527.244} C_VEL
LIN {X 0,Y 471.013,Z 350.922,A -85,B 0,C 180,E1 22523.852,E2 22523.852} C_VEL
LIN {X 0,Y 470.856,Z 396.275,A -85,B 0,C 180,E1 22520.64,E2 22520.64} C_VEL
LIN {X 0,Y 470.244,Z 444.311,A -85,B 0,C 180,E1 22517.126,E2 22517.126} C_VEL
LIN {X 0,Y 469.427,Z 491.959,A -85,B 0,C 180,E1 22513.55,E2 22513.55} C_VEL
LIN {X 0,Y 468.995,Z 500.24,A -85,B 0,C 180,E1 22512.935,E2 22512.935} C_VEL
LIN {X 0,Y 468.42,Z 504.528,A -85,B 0,C 180,E1 22512.677,E2 22512.677} C_VEL
LIN {X 0,Y 467.392,Z 617.48,A -85,B 0,C 180,E1 22510.73,E2 22510.73} C_VEL
LIN {X 0,Y 467.361,Z 632.758,A -85,B 0,C 180,E1 22510.225,E2 22510.225} C_VEL
LIN {X 0,Y 467.215,Z 646.344,A -85,B 0,C 180,E1 22509.546,E2 22509.546} C_VEL
LIN {X 0,Y 466.956,Z 659.117,A -85,B 0,C 180,E1 22508.682,E2 22508.682} C_VEL
LIN {X 0,Y 466.635,Z 671.569,A -85,B 0,C 180,E1 22507.572,E2 22507.572} C_VEL
LIN {X 0,Y 466.264,Z 682.727,A -85,B 0,C 180,E1 22506.278,E2 22506.278} C_VEL
LIN {X 0,Y 465.926,Z 691.815,A -85,B 0,C 180,E1 22504.924,E2 22504.924} C_VEL
LIN {X 0,Y 465.615,Z 699.567,A -85,B 0,C 180,E1 22503.447,E2 22503.447} C_VEL
LIN {X 0,Y 465.339,Z 706.313,A -85,B 0,C 180,E1 22501.723,E2 22501.723} C_VEL
LIN {X 0,Y 465.138,Z 711.252,A -85,B 0,C 180,E1 22499.876,E2 22499.876} C_VEL
LIN {X 0,Y 465.011,Z 714.107,A -85,B 0,C 180,E1 22498.028,E2 22498.028} C_VEL
LIN {X 0,Y 464.94,Z 715.046,A -85,B 0,C 180,E1 22496.177,E2 22496.177} C_VEL
LIN {X 0,Y 464.924,Z 714.236,A -85,B 0,C 180,E1 22494.446,E2 22494.446} C_VEL
LIN {X 0,Y 464.965,Z 711.534,A -85,B 0,C 180,E1 22492.586,E2 22492.586} C_VEL
LIN {X 0,Y 465.08,Z 706.793,A -85,B 0,C 180,E1 22490.721,E2 22490.721} C_VEL
LIN {X 0,Y 465.274,Z 700.273,A -85,B 0,C 180,E1 22488.973,E2 22488.973} C_VEL
LIN {X 0,Y 465.556,Z 692.067,A -85,B 0,C 180,E1 22487.346,E2 22487.346} C_VEL
LIN {X 0,Y 465.87,Z 683.008,A -85,B 0,C 180,E1 22485.954,E2 22485.954} C_VEL
LIN {X 0,Y 466.236,Z 672.186,A -85,B 0,C 180,E1 22484.641,E2 22484.641} C_VEL
LIN {X 0,Y 466.615,Z 659.443,A -85,B 0,C 180,E1 22483.441,E2 22483.441} C_VEL
LIN {X 0,Y 466.979,Z 645.195,A -85,B 0,C 180,E1 22482.428,E2 22482.428} C_VEL
LIN {X 0,Y 467.219,Z 630.341,A -85,B 0,C 180,E1 22481.664,E2 22481.664} C_VEL
LIN {X 0,Y 467.346,Z 614.646,A -85,B 0,C 180,E1 22481.131,E2 22481.131} C_VEL
LIN {X 0,Y 467.458,Z 586.453,A -85,B 0,C 180,E1 22480.631,E2 22480.631} C_VEL
LIN {X 0,Y 468.411,Z 497.563,A -85,B 0,C 180,E1 22479.152,E2 22479.152} C_VEL
LIN {X 0,Y 469.472,Z 453.562,A -85,B 0,C 180,E1 22475.719,E2 22475.719} C_VEL
LIN {X 0,Y 470.611,Z 407.301,A -85,B 0,C 180,E1 22472.109,E2 22472.109} C_VEL
LIN {X 0,Y 471.62,Z 362.851,A -85,B 0,C 180,E1 22468.636,E2 22468.636} C_VEL
LIN {X 0,Y 472.496,Z 320.319,A -85,B 0,C 180,E1 22465.302,E2 22465.302} C_VEL
LIN {X 0,Y 473.15,Z 280.019,A -85,B 0,C 180,E1 22462.168,E2 22462.168} C_VEL
LIN {X 0,Y 467.354,Z 262.091,A -85,B 0,C 180,E1 22460.355,E2 22460.355} C_VEL
LIN {X 0,Y 468.634,Z 262.678,A -85,B 0,C 180,E1 22459.992,E2 22459.992} C_VEL
LIN {X 0,Y 470.187,Z 265.384,A -85,B 0,C 180,E1 22459.243,E2 22459.243} C_VEL
LIN {X 0,Y 472.544,Z 270.113,A -85,B 0,C 180,E1 22458.038,E2 22458.038} C_VEL
LIN {X 0,Y 473.424,Z 272.003,A -85,B 0,C 180,E1 22457.581,E2 22457.581} C_VEL
LIN {X 0,Y 474.406,Z 275.326,A -85,B 0,C 180,E1 22456.896,E2 22456.896} C_VEL
LIN {X 0,Y 474.407,Z 282.356,A -85,B 0,C 180,E1 22455.846,E2 22455.846} C_VEL
LIN {X 0,Y 474.376,Z 290.268,A -85,B 0,C 180,E1 22454.693,E2 22454.693} C_VEL
LIN {X 0,Y 475.163,Z 293.262,A -85,B 0,C 180,E1 22454.129,E2 22454.129} C_VEL
LIN {X 0,Y 480.836,Z 306.878,A -85,B 0,C 180,E1 22451.351,E2 22451.351} C_VEL
LIN {X 0,Y 481.225,Z 308.19,A -85,B 0,C 180,E1 22451.118,E2 22451.118} C_VEL
LIN {X 0,Y 479.135,Z 325.617,A -85,B 0,C 180,E1 22449.213,E2 22449.213} C_VEL
LIN {X 0,Y 480.097,Z 330.43,A -85,B 0,C 180,E1 22449.027,E2 22449.027} C_VEL
LIN {X 0,Y 477.85,Z 417.493,A -85,B 0,C 180,E1 22447.527,E2 22447.527} C_VEL
LIN {X 0,Y 473.959,Z 524.383,A -85,B 0,C 180,E1 22445.456,E2 22445.456} C_VEL
LIN {X 0,Y 472.049,Z 574.963,A -85,B 0,C 180,E1 22444.376,E2 22444.376} C_VEL
LIN {X 0,Y 471.038,Z 595.18,A -85,B 0,C 180,E1 22443.716,E2 22443.716} C_VEL
LIN {X 0,Y 469.692,Z 615.758,A -85,B 0,C 180,E1 22442.804,E2 22442.804} C_VEL
LIN {X 0,Y 468.156,Z 635.226,A -85,B 0,C 180,E1 22441.695,E2 22441.695} C_VEL
LIN {X 0,Y 466.486,Z 653.799,A -85,B 0,C 180,E1 22440.387,E2 22440.387} C_VEL
LIN {X 0,Y 464.774,Z 671.458,A -85,B 0,C 180,E1 22438.886,E2 22438.886} C_VEL
LIN {X 0,Y 463.114,Z 687.651,A -85,B 0,C 180,E1 22437.24,E2 22437.24} C_VEL
LIN {X 0,Y 461.488,Z 703.04,A -85,B 0,C 180,E1 22435.38,E2 22435.38} C_VEL
LIN {X 0,Y 460.063,Z 716.608,A -85,B 0,C 180,E1 22433.436,E2 22433.436} C_VEL
LIN {X 0,Y 458.823,Z 728.94,A -85,B 0,C 180,E1 22431.342,E2 22431.342} C_VEL
LIN {X 0,Y 457.816,Z 739.88,A -85,B 0,C 180,E1 22429.123,E2 22429.123} C_VEL
LIN {X 0,Y 457.048,Z 749.417,A -85,B 0,C 180,E1 22426.785,E2 22426.785} C_VEL
LIN {X 0,Y 456.501,Z 757.451,A -85,B 0,C 180,E1 22424.33,E2 22424.33} C_VEL
LIN {X 0,Y 456.195,Z 763.683,A -85,B 0,C 180,E1 22421.89,E2 22421.89} C_VEL
LIN {X 0,Y 456.027,Z 768.51,A -85,B 0,C 180,E1 22419.338,E2 22419.338} C_VEL
LIN {X 0,Y 455.971,Z 771.682,A -85,B 0,C 180,E1 22416.801,E2 22416.801} C_VEL
LIN {X 0,Y 455.948,Z 773.301,A -85,B 0,C 180,E1 22414.15,E2 22414.15} C_VEL
LIN {X 0,Y 455.944,Z 773.266,A -85,B 0,C 180,E1 22411.634,E2 22411.634} C_VEL
LIN {X 0,Y 455.963,Z 771.685,A -85,B 0,C 180,E1 22409.121,E2 22409.121} C_VEL
LIN {X 0,Y 456.024,Z 768.553,A -85,B 0,C 180,E1 22406.606,E2 22406.606} C_VEL
LIN {X 0,Y 456.188,Z 763.829,A -85,B 0,C 180,E1 22404.087,E2 22404.087} C_VEL
LIN {X 0,Y 456.489,Z 757.768,A -85,B 0,C 180,E1 22401.688,E2 22401.688} C_VEL
LIN {X 0,Y 457.036,Z 749.505,A -85,B 0,C 180,E1 22399.156,E2 22399.156} C_VEL
LIN {X 0,Y 457.83,Z 739.666,A -85,B 0,C 180,E1 22396.743,E2 22396.743} C_VEL
LIN {X 0,Y 458.885,Z 728.31,A -85,B 0,C 180,E1 22394.454,E2 22394.454} C_VEL
LIN {X 0,Y 460.096,Z 716.227,A -85,B 0,C 180,E1 22392.418,E2 22392.418} C_VEL
LIN {X 0,Y 461.541,Z 702.433,A -85,B 0,C 180,E1 22390.454,E2 22390.454} C_VEL
LIN {X 0,Y 463.173,Z 687.021,A -85,B 0,C 180,E1 22388.603,E2 22388.603} C_VEL
LIN {X 0,Y 464.759,Z 671.673,A -85,B 0,C 180,E1 22387.041,E2 22387.041} C_VEL
LIN {X 0,Y 466.451,Z 654.375,A -85,B 0,C 180,E1 22385.562,E2 22385.562} C_VEL
LIN {X 0,Y 468.138,Z 635.486,A -85,B 0,C 180,E1 22384.231,E2 22384.231} C_VEL
LIN {X 0,Y 469.657,Z 616.131,A -85,B 0,C 180,E1 22383.129,E2 22383.129} C_VEL
LIN {X 0,Y 470.972,Z 595.63,A -85,B 0,C 180,E1 22382.218,E2 22382.218} C_VEL
LIN {X 0,Y 472.001,Z 574.749,A -85,B 0,C 180,E1 22381.539,E2 22381.539} C_VEL
LIN {X 0,Y 473.659,Z 529.245,A -85,B 0,C 180,E1 22380.573,E2 22380.573} C_VEL
LIN {X 0,Y 477.561,Z 419.304,A -85,B 0,C 180,E1 22378.458,E2 22378.458} C_VEL
LIN {X 0,Y 479.813,Z 329.549,A -85,B 0,C 180,E1 22376.92,E2 22376.92} C_VEL
LIN {X 0,Y 479.659,Z 324.832,A -85,B 0,C 180,E1 22376.819,E2 22376.819} C_VEL
LIN {X 0,Y 479.327,Z 322.825,A -85,B 0,C 180,E1 22376.728,E2 22376.728} C_VEL
LIN {X 0,Y 480.92,Z 305.581,A -85,B 0,C 180,E1 22375.151,E2 22375.151} C_VEL
LIN {X 0,Y 473.486,Z 289.187,A -85,B 0,C 180,E1 22372.363,E2 22372.363} C_VEL
LIN {X 0,Y 467.71,Z 277.144,A -85,B 0,C 180,E1 22370.127,E2 22370.127} C_VEL
LIN {X 0,Y 463.494,Z 268.806,A -85,B 0,C 180,E1 22368.466,E2 22368.466} C_VEL
LIN {X 0,Y 461.462,Z 264.759,A -85,B 0,C 180,E1 22367.634,E2 22367.634} C_VEL
LIN {X 0,Y 459.754,Z 261.431,A -85,B 0,C 180,E1 22366.931,E2 22366.931} C_VEL
LIN {X 0,Y 458.718,Z 259.747,A -85,B 0,C 180,E1 22366.539,E2 22366.539} C_VEL
LIN {X 0,Y 457.17,Z 256.383,A -85,B 0,C 180,E1 22365.837,E2 22365.837} C_VEL
LIN {X 0,Y 457.069,Z 255.801,A -85,B 0,C 180,E1 22365.671,E2 22365.671} C_VEL
LIN {X 0,Y 457.063,Z 255.796,A -85,B 0,C 180,E1 22361.946,E2 22361.946} C_VEL
LIN {X 0,Y 457.081,Z 255.797,A -85,B 0,C 180,E1 22358.248,E2 22358.248} C_VEL
LIN {X 0,Y 457.065,Z 255.803,A -85,B 0,C 180,E1 22354.44,E2 22354.44} C_VEL
LIN {X 0,Y 457.08,Z 255.825,A -85,B 0,C 180,E1 22352.501,E2 22352.501} C_VEL
LIN {X 0,Y 465.816,Z 282.659,A -85,B 0,C 180,E1 22349.584,E2 22349.584} C_VEL
LIN {X 0,Y 466.215,Z 285.131,A -85,B 0,C 180,E1 22349.344,E2 22349.344} C_VEL
LIN {X 0,Y 465.337,Z 327.67,A -85,B 0,C 180,E1 22345.724,E2 22345.724} C_VEL
LIN {X 0,Y 464.346,Z 369.336,A -85,B 0,C 180,E1 22342.194,E2 22342.194} C_VEL
LIN {X 0,Y 463.16,Z 412.884,A -85,B 0,C 180,E1 22338.503,E2 22338.503} C_VEL
LIN {X 0,Y 462.244,Z 449.28,A -85,B 0,C 180,E1 22335.454,E2 22335.454} C_VEL
LIN {X 0,Y 462.115,Z 475.581,A -85,B 0,C 180,E1 22334.982,E2 22334.982} C_VEL
LIN {X 0,Y 460.744,Z 592.89,A -85,B 0,C 180,E1 22332.952,E2 22332.952} C_VEL
LIN {X 0,Y 460.582,Z 609.256,A -85,B 0,C 180,E1 22332.443,E2 22332.443} C_VEL
LIN {X 0,Y 460.244,Z 624.888,A -85,B 0,C 180,E1 22331.72,E2 22331.72} C_VEL
LIN {X 0,Y 459.82,Z 640.073,A -85,B 0,C 180,E1 22330.778,E2 22330.778} C_VEL
LIN {X 0,Y 459.289,Z 654.726,A -85,B 0,C 180,E1 22329.587,E2 22329.587} C_VEL
LIN {X 0,Y 458.793,Z 666.932,A -85,B 0,C 180,E1 22328.341,E2 22328.341} C_VEL
LIN {X 0,Y 458.258,Z 679.257,A -85,B 0,C 180,E1 22326.767,E2 22326.767} C_VEL
LIN {X 0,Y 457.81,Z 689.347,A -85,B 0,C 180,E1 22325.138,E2 22325.138} C_VEL
LIN {X 0,Y 457.476,Z 697.987,A -85,B 0,C 180,E1 22323.384,E2 22323.384} C_VEL
LIN {X 0,Y 457.232,Z 705.007,A -85,B 0,C 180,E1 22321.504,E2 22321.504} C_VEL
LIN {X 0,Y 457.092,Z 710.195,A -85,B 0,C 180,E1 22319.624,E2 22319.624} C_VEL
LIN {X 0,Y 457.022,Z 713.769,A -85,B 0,C 180,E1 22317.618,E2 22317.618} C_VEL
LIN {X 0,Y 457.019,Z 715.518,A -85,B 0,C 180,E1 22315.735,E2 22315.735} C_VEL
LIN {X 0,Y 457.08,Z 715.573,A -85,B 0,C 180,E1 22313.721,E2 22313.721} C_VEL
LIN {X 0,Y 457.18,Z 714.015,A -85,B 0,C 180,E1 22311.828,E2 22311.828} C_VEL
LIN {X 0,Y 457.366,Z 710.431,A -85,B 0,C 180,E1 22309.801,E2 22309.801} C_VEL
LIN {X 0,Y 457.603,Z 705.634,A -85,B 0,C 180,E1 22308.02,E2 22308.02} C_VEL
LIN {X 0,Y 457.901,Z 698.948,A -85,B 0,C 180,E1 22306.231,E2 22306.231} C_VEL
LIN {X 0,Y 458.304,Z 690.849,A -85,B 0,C 180,E1 22304.564,E2 22304.564} C_VEL
LIN {X 0,Y 458.746,Z 681.229,A -85,B 0,C 180,E1 22303.019,E2 22303.019} C_VEL
LIN {X 0,Y 459.223,Z 670.176,A -85,B 0,C 180,E1 22301.597,E2 22301.597} C_VEL
LIN {X 0,Y 459.691,Z 657.395,A -85,B 0,C 180,E1 22300.298,E2 22300.298} C_VEL
LIN {X 0,Y 460.073,Z 644.461,A -85,B 0,C 180,E1 22299.253,E2 22299.253} C_VEL
LIN {X 0,Y 460.384,Z 629.58,A -85,B 0,C 180,E1 22298.334,E2 22298.334} C_VEL
LIN {X 0,Y 460.569,Z 614.131,A -85,B 0,C 180,E1 22297.633,E2 22297.633} C_VEL
LIN {X 0,Y 460.593,Z 597.082,A -85,B 0,C 180,E1 22297.122,E2 22297.122} C_VEL
LIN {X 0,Y 461.793,Z 489.911,A -85,B 0,C 180,E1 22295.228,E2 22295.228} C_VEL
LIN {X 0,Y 462.367,Z 459.143,A -85,B 0,C 180,E1 22294.649,E2 22294.649} C_VEL
LIN {X 0,Y 463.597,Z 451.208,A -85,B 0,C 180,E1 22294.075,E2 22294.075} C_VEL
LIN {X 0,Y 464.196,Z 412.333,A -85,B 0,C 180,E1 22290.987,E2 22290.987} C_VEL
LIN {X 0,Y 464.486,Z 377.669,A -85,B 0,C 180,E1 22288.316,E2 22288.316} C_VEL
LIN {X 0,Y 464.417,Z 342.766,A -85,B 0,C 180,E1 22285.738,E2 22285.738} C_VEL
LIN {X 0,Y 464.402,Z 340.691,A -85,B 0,C 180,E1 22285.587,E2 22285.587} C_VEL
LIN {X 0,Y 465.877,Z 341.425,A -85,B 0,C 180,E1 22285.338,E2 22285.338} C_VEL
LIN {X 0,Y 468.316,Z 341.085,A -85,B 0,C 180,E1 22285.07,E2 22285.07} C_VEL
LIN {X 0,Y 470.772,Z 340.079,A -85,B 0,C 180,E1 22284.861,E2 22284.861} C_VEL
LIN {X 0,Y 474.67,Z 339.437,A -85,B 0,C 180,E1 22284.453,E2 22284.453} C_VEL
LIN {X 0,Y 477.156,Z 338.736,A -85,B 0,C 180,E1 22284.223,E2 22284.223} C_VEL
LIN {X 0,Y 483.383,Z 337.447,A -85,B 0,C 180,E1 22283.621,E2 22283.621} C_VEL
LIN {X 0,Y 482.996,Z 356.841,A -85,B 0,C 180,E1 22282.061,E2 22282.061} C_VEL
LIN {X 0,Y 484.496,Z 374.085,A -85,B 0,C 180,E1 22280.519,E2 22280.519} C_VEL
LIN {X 0,Y 487.761,Z 389.332,A -85,B 0,C 180,E1 22279.008,E2 22279.008} C_VEL
LIN {X 0,Y 492.629,Z 402.526,A -85,B 0,C 180,E1 22277.558,E2 22277.558} C_VEL
LIN {X 0,Y 499.153,Z 414.276,A -85,B 0,C 180,E1 22276.126,E2 22276.126} C_VEL
LIN {X 0,Y 507.612,Z 424.888,A -85,B 0,C 180,E1 22274.678,E2 22274.678} C_VEL
LIN {X 0,Y 517.068,Z 433.425,A -85,B 0,C 180,E1 22273.351,E2 22273.351} C_VEL
LIN {X 0,Y 528.012,Z 440.564,A -85,B 0,C 180,E1 22272.073,E2 22272.073} C_VEL
LIN {X 0,Y 537.643,Z 445.384,A -85,B 0,C 180,E1 22271.099,E2 22271.099} C_VEL
LIN {X 0,Y 515.992,Z 478.341,A -85,B 0,C 180,E1 22270.401,E2 22270.401} C_VEL
LIN {X 0,Y 505.57,Z 496.567,A -85,B 0,C 180,E1 22269.885,E2 22269.885} C_VEL
LIN {X 0,Y 498.515,Z 511.748,A -85,B 0,C 180,E1 22269.331,E2 22269.331} C_VEL
LIN {X 0,Y 495.933,Z 517.266,A -85,B 0,C 180,E1 22269.128,E2 22269.128} C_VEL
LIN {X 0,Y 488.852,Z 531.881,A -85,B 0,C 180,E1 22268.596,E2 22268.596} C_VEL
LIN {X 0,Y 479.867,Z 556.496,A -85,B 0,C 180,E1 22267.508,E2 22267.508} C_VEL
LIN {X 0,Y 478.72,Z 572.944,A -85,B 0,C 180,E1 22267.305,E2 22267.305} C_VEL
LIN {X 0,Y 477.856,Z 603.94,A -85,B 0,C 180,E1 22266.747,E2 22266.747} C_VEL
LIN {X 0,Y 476.479,Z 627.664,A -85,B 0,C 180,E1 22266.116,E2 22266.116} C_VEL
LIN {X 0,Y 474.886,Z 650.21,A -85,B 0,C 180,E1 22265.29,E2 22265.29} C_VEL
LIN {X 0,Y 473.006,Z 672.975,A -85,B 0,C 180,E1 22264.214,E2 22264.214} C_VEL
LIN {X 0,Y 471.085,Z 693.897,A -85,B 0,C 180,E1 22262.985,E2 22262.985} C_VEL
LIN {X 0,Y 469.144,Z 713.174,A -85,B 0,C 180,E1 22261.62,E2 22261.62} C_VEL
LIN {X 0,Y 467.153,Z 731.854,A -85,B 0,C 180,E1 22260.056,E2 22260.056} C_VEL
LIN {X 0,Y 465.15,Z 749.786,A -85,B 0,C 180,E1 22258.293,E2 22258.293} C_VEL
LIN {X 0,Y 463.04,Z 768.283,A -85,B 0,C 180,E1 22256.136,E2 22256.136} C_VEL
LIN {X 0,Y 461.128,Z 785.244,A -85,B 0,C 180,E1 22253.785,E2 22253.785} C_VEL
LIN {X 0,Y 459.799,Z 797.066,A -85,B 0,C 180,E1 22251.83,E2 22251.83} C_VEL
LIN {X 0,Y 458.457,Z 809.736,A -85,B 0,C 180,E1 22249.36,E2 22249.36} C_VEL
LIN {X 0,Y 457.384,Z 821.408,A -85,B 0,C 180,E1 22246.641,E2 22246.641} C_VEL
LIN {X 0,Y 456.646,Z 831.353,A -85,B 0,C 180,E1 22243.808,E2 22243.808} C_VEL
LIN {X 0,Y 456.211,Z 839.356,A -85,B 0,C 180,E1 22240.931,E2 22240.931} C_VEL
LIN {X 0,Y 456.012,Z 845.389,A -85,B 0,C 180,E1 22238.067,E2 22238.067} C_VEL
LIN {X 0,Y 455.931,Z 849.439,A -85,B 0,C 180,E1 22235.285,E2 22235.285} C_VEL
LIN {X 0,Y 455.909,Z 851.714,A -85,B 0,C 180,E1 22232.64,E2 22232.64} C_VEL
LIN {X 0,Y 455.912,Z 852.5,A -85,B 0,C 180,E1 22230,E2 22230} C_VEL
LIN {X 0,Y 455.911,Z 851.645,A -85,B 0,C 180,E1 22227.234,E2 22227.234} C_VEL
LIN {X 0,Y 455.933,Z 849.286,A -85,B 0,C 180,E1 22224.589,E2 22224.589} C_VEL
LIN {X 0,Y 456.012,Z 845.388,A -85,B 0,C 180,E1 22221.933,E2 22221.933} C_VEL
LIN {X 0,Y 456.211,Z 839.356,A -85,B 0,C 180,E1 22219.069,E2 22219.069} C_VEL
LIN {X 0,Y 456.646,Z 831.352,A -85,B 0,C 180,E1 22216.192,E2 22216.192} C_VEL
LIN {X 0,Y 457.384,Z 821.408,A -85,B 0,C 180,E1 22213.359,E2 22213.359} C_VEL
LIN {X 0,Y 458.455,Z 809.736,A -85,B 0,C 180,E1 22210.64,E2 22210.64} C_VEL
LIN {X 0,Y 459.882,Z 796.351,A -85,B 0,C 180,E1 22208.04,E2 22208.04} C_VEL
LIN {X 0,Y 461.224,Z 784.359,A -85,B 0,C 180,E1 22206.084,E2 22206.084} C_VEL
LIN {X 0,Y 463.036,Z 768.246,A -85,B 0,C 180,E1 22203.863,E2 22203.863} C_VEL
LIN {X 0,Y 465.01,Z 750.863,A -85,B 0,C 180,E1 22201.832,E2 22201.832} C_VEL
LIN {X 0,Y 467.146,Z 731.788,A -85,B 0,C 180,E1 22199.944,E2 22199.944} C_VEL
LIN {X 0,Y 469.213,Z 712.183,A -85,B 0,C 180,E1 22198.313,E2 22198.313} C_VEL
LIN {X 0,Y 471.37,Z 690.662,A -85,B 0,C 180,E1 22196.82,E2 22196.82} C_VEL
LIN {X 0,Y 473.252,Z 669.303,A -85,B 0,C 180,E1 22195.61,E2 22195.61} C_VEL
LIN {X 0,Y 475.054,Z 647.016,A -85,B 0,C 180,E1 22194.596,E2 22194.596} C_VEL
LIN {X 0,Y 476.659,Z 623.357,A -85,B 0,C 180,E1 22193.767,E2 22193.767} C_VEL
LIN {X 0,Y 478.036,Z 598.422,A -85,B 0,C 180,E1 22193.151,E2 22193.151} C_VEL
LIN {X 0,Y 479.025,Z 565.85,A -85,B 0,C 180,E1 22192.612,E2 22192.612} C_VEL
LIN {X 0,Y 480.182,Z 556.33,A -85,B 0,C 180,E1 22192.516,E2 22192.516} C_VEL
LIN {X 0,Y 490.287,Z 534.342,A -85,B 0,C 180,E1 22191.388,E2 22191.388} C_VEL
LIN {X 0,Y 498.096,Z 521.341,A -85,B 0,C 180,E1 22190.852,E2 22190.852} C_VEL
LIN {X 0,Y 501.409,Z 516.022,A -85,B 0,C 180,E1 22190.645,E2 22190.645} C_VEL
LIN {X 0,Y 509.098,Z 502.937,A -85,B 0,C 180,E1 22190.115,E2 22190.115} C_VEL
LIN {X 0,Y 520.185,Z 487.415,A -85,B 0,C 180,E1 22189.627,E2 22189.627} C_VEL
LIN {X 0,Y 528.745,Z 476.384,A -85,B 0,C 180,E1 22189.334,E2 22189.334} C_VEL
LIN {X 0,Y 516.413,Z 469.569,A -85,B 0,C 180,E1 22188.029,E2 22188.029} C_VEL
LIN {X 0,Y 505.913,Z 461.375,A -85,B 0,C 180,E1 22186.66,E2 22186.66} C_VEL
LIN {X 0,Y 497.21,Z 451.906,A -85,B 0,C 180,E1 22185.223,E2 22185.223} C_VEL
LIN {X 0,Y 490.587,Z 441.829,A -85,B 0,C 180,E1 22183.822,E2 22183.822} C_VEL
LIN {X 0,Y 485.219,Z 429.759,A -85,B 0,C 180,E1 22182.288,E2 22182.288} C_VEL
LIN {X 0,Y 481.672,Z 416.4,A -85,B 0,C 180,E1 22180.74,E2 22180.74} C_VEL
LIN {X 0,Y 479.765,Z 400.737,A -85,B 0,C 180,E1 22179.081,E2 22179.081} C_VEL
LIN {X 0,Y 479.816,Z 383.29,A -85,B 0,C 180,E1 22177.404,E2 22177.404} C_VEL
LIN {X 0,Y 484.894,Z 333.262,A -85,B 0,C 180,E1 22172.939,E2 22172.939} C_VEL
LIN {X 0,Y 486.774,Z 315.711,A -85,B 0,C 180,E1 22171.31,E2 22171.31} C_VEL
LIN {X 0,Y 481.604,Z 304.421,A -85,B 0,C 180,E1 22169.311,E2 22169.311} C_VEL
LIN {X 0,Y 473.318,Z 307.236,A -85,B 0,C 180,E1 22168.379,E2 22168.379} C_VEL
LIN {X 0,Y 469.575,Z 308.448,A -85,B 0,C 180,E1 22167.933,E2 22167.933} C_VEL
LIN {X 0,Y 468.498,Z 308.738,A -85,B 0,C 180,E1 22167.795,E2 22167.795} C_VEL
LIN {X 0,Y 465.399,Z 310.15,A -85,B 0,C 180,E1 22167.465,E2 22167.465} C_VEL
LIN {X 0,Y 463.421,Z 310.001,A -85,B 0,C 180,E1 22167.098,E2 22167.098} C_VEL
LIN {X 0,Y 463.655,Z 354.387,A -85,B 0,C 180,E1 22164.052,E2 22164.052} C_VEL
LIN {X 0,Y 463.424,Z 394.349,A -85,B 0,C 180,E1 22161.192,E2 22161.192} C_VEL
LIN {X 0,Y 462.958,Z 434.85,A -85,B 0,C 180,E1 22158.249,E2 22158.249} C_VEL
LIN {X 0,Y 462.169,Z 480.022,A -85,B 0,C 180,E1 22154.854,E2 22154.854} C_VEL
LIN {X 0,Y 461.66,Z 500.185,A -85,B 0,C 180,E1 22153.335,E2 22153.335} C_VEL
LIN {X 0,Y 460.789,Z 506.167,A -85,B 0,C 180,E1 22152.954,E2 22152.954} C_VEL
LIN {X 0,Y 459.664,Z 618.482,A -85,B 0,C 180,E1 22150.964,E2 22150.964} C_VEL
LIN {X 0,Y 459.642,Z 633.326,A -85,B 0,C 180,E1 22150.475,E2 22150.475} C_VEL
LIN {X 0,Y 459.516,Z 646.375,A -85,B 0,C 180,E1 22149.834,E2 22149.834} C_VEL
LIN {X 0,Y 459.248,Z 659.53,A -85,B 0,C 180,E1 22148.955,E2 22148.955} C_VEL
LIN {X 0,Y 458.908,Z 672.226,A -85,B 0,C 180,E1 22147.826,E2 22147.826} C_VEL
LIN {X 0,Y 458.546,Z 682.608,A -85,B 0,C 180,E1 22146.636,E2 22146.636} C_VEL
LIN {X 0,Y 458.182,Z 692.091,A -85,B 0,C 180,E1 22145.258,E2 22145.258} C_VEL
LIN {X 0,Y 457.815,Z 700.69,A -85,B 0,C 180,E1 22143.631,E2 22143.631} C_VEL
LIN {X 0,Y 457.505,Z 707.506,A -85,B 0,C 180,E1 22141.878,E2 22141.878} C_VEL
LIN {X 0,Y 457.28,Z 712.501,A -85,B 0,C 180,E1 22140,E2 22140} C_VEL
LIN {X 0,Y 457.134,Z 715.401,A -85,B 0,C 180,E1 22138.119,E2 22138.119} C_VEL
LIN {X 0,Y 457.059,Z 716.372,A -85,B 0,C 180,E1 22136.362,E2 22136.362} C_VEL
LIN {X 0,Y 457.033,Z 715.593,A -85,B 0,C 180,E1 22134.476,E2 22134.476} C_VEL
LIN {X 0,Y 457.075,Z 712.894,A -85,B 0,C 180,E1 22132.584,E2 22132.584} C_VEL
LIN {X 0,Y 457.194,Z 708.147,A -85,B 0,C 180,E1 22130.686,E2 22130.686} C_VEL
LIN {X 0,Y 457.399,Z 701.614,A -85,B 0,C 180,E1 22128.909,E2 22128.909} C_VEL
LIN {X 0,Y 457.666,Z 694.108,A -85,B 0,C 180,E1 22127.38,E2 22127.38} C_VEL
LIN {X 0,Y 457.994,Z 685.332,A -85,B 0,C 180,E1 22125.976,E2 22125.976} C_VEL
LIN {X 0,Y 458.391,Z 674.082,A -85,B 0,C 180,E1 22124.567,E2 22124.567} C_VEL
LIN {X 0,Y 458.785,Z 661.479,A -85,B 0,C 180,E1 22123.346,E2 22123.346} C_VEL
LIN {X 0,Y 459.131,Z 648.468,A -85,B 0,C 180,E1 22122.379,E2 22122.379} C_VEL
LIN {X 0,Y 459.393,Z 634.462,A -85,B 0,C 180,E1 22121.603,E2 22121.603} C_VEL
LIN {X 0,Y 459.548,Z 619.609,A -85,B 0,C 180,E1 22121.034,E2 22121.034} C_VEL
LIN {X 0,Y 459.567,Z 602.986,A -85,B 0,C 180,E1 22120.668,E2 22120.668} C_VEL
LIN {X 0,Y 460.732,Z 498.41,A -85,B 0,C 180,E1 22118.884,E2 22118.884} C_VEL
LIN {X 0,Y 461.84,Z 455.379,A -85,B 0,C 180,E1 22115.506,E2 22115.506} C_VEL
LIN {X 0,Y 463.05,Z 408.846,A -85,B 0,C 180,E1 22111.848,E2 22111.848} C_VEL
LIN {X 0,Y 464.138,Z 363.602,A -85,B 0,C 180,E1 22108.289,E2 22108.289} C_VEL
LIN {X 0,Y 465.089,Z 320.63,A -85,B 0,C 180,E1 22104.894,E2 22104.894} C_VEL
LIN {X 0,Y 465.747,Z 282.408,A -85,B 0,C 180,E1 22101.888,E2 22101.888} C_VEL
LIN {X 0,Y 461.4,Z 268.79,A -85,B 0,C 180,E1 22100.504,E2 22100.504} C_VEL
LIN {X 0,Y 463.033,Z 269.082,A -85,B 0,C 180,E1 22100.108,E2 22100.108} C_VEL
LIN {X 0,Y 463.713,Z 269.186,A -85,B 0,C 180,E1 22099.948,E2 22099.948} C_VEL
LIN {X 0,Y 465.127,Z 272.019,A -85,B 0,C 180,E1 22099.194,E2 22099.194} C_VEL
LIN {X 0,Y 467.223,Z 276.201,A -85,B 0,C 180,E1 22098.111,E2 22098.111} C_VEL
LIN {X 0,Y 471.236,Z 284.654,A -85,B 0,C 180,E1 22096.066,E2 22096.066} C_VEL
LIN {X 0,Y 475.163,Z 293.262,A -85,B 0,C 180,E1 22094.129,E2 22094.129} C_VEL
LIN {X 0,Y 476.208,Z 297.525,A -85,B 0,C 180,E1 22093.354,E2 22093.354} C_VEL
LIN {X 0,Y 476.146,Z 304.157,A -85,B 0,C 180,E1 22092.444,E2 22092.444} C_VEL
LIN {X 0,Y 474.332,Z 317.342,A -85,B 0,C 180,E1 22090.942,E2 22090.942} C_VEL
LIN {X 0,Y 473.085,Z 328.015,A -85,B 0,C 180,E1 22089.782,E2 22089.782} C_VEL
LIN {X 0,Y 473.91,Z 332.347,A -85,B 0,C 180,E1 22089.614,E2 22089.614} C_VEL
LIN {X 0,Y 471.594,Z 417.004,A -85,B 0,C 180,E1 22088.139,E2 22088.139} C_VEL
LIN {X 0,Y 467.812,Z 513.774,A -85,B 0,C 180,E1 22086.231,E2 22086.231} C_VEL
LIN {X 0,Y 465.234,Z 575.635,A -85,B 0,C 180,E1 22084.882,E2 22084.882} C_VEL
LIN {X 0,Y 464.129,Z 596.231,A -85,B 0,C 180,E1 22084.194,E2 22084.194} C_VEL
LIN {X 0,Y 462.723,Z 616.274,A -85,B 0,C 180,E1 22083.288,E2 22083.288} C_VEL
LIN {X 0,Y 461.09,Z 635.66,A -85,B 0,C 180,E1 22082.165,E2 22082.165} C_VEL
LIN {X 0,Y 459.3,Z 654.142,A -85,B 0,C 180,E1 22080.842,E2 22080.842} C_VEL
LIN {X 0,Y 457.434,Z 672.005,A -85,B 0,C 180,E1 22079.291,E2 22079.291} C_VEL
LIN {X 0,Y 455.621,Z 688.456,A -85,B 0,C 180,E1 22077.584,E2 22077.584} C_VEL
LIN {X 0,Y 453.915,Z 703.656,A -85,B 0,C 180,E1 22075.718,E2 22075.718} C_VEL
LIN {X 0,Y 452.392,Z 717.408,A -85,B 0,C 180,E1 22073.719,E2 22073.719} C_VEL
LIN {X 0,Y 451.078,Z 729.754,A -85,B 0,C 180,E1 22071.59,E2 22071.59} C_VEL
LIN {X 0,Y 450.004,Z 740.716,A -85,B 0,C 180,E1 22069.333,E2 22069.333} C_VEL
LIN {X 0,Y 449.183,Z 750.258,A -85,B 0,C 180,E1 22066.954,E2 22066.954} C_VEL
LIN {X 0,Y 448.572,Z 758.676,A -85,B 0,C 180,E1 22064.325,E2 22064.325} C_VEL
LIN {X 0,Y 448.232,Z 765.151,A -85,B 0,C 180,E1 22061.685,E2 22061.685} C_VEL
LIN {X 0,Y 448.065,Z 769.704,A -85,B 0,C 180,E1 22059.116,E2 22059.116} C_VEL
LIN {X 0,Y 447.997,Z 772.659,A -85,B 0,C 180,E1 22056.536,E2 22056.536} C_VEL
LIN {X 0,Y 447.979,Z 774.073,A -85,B 0,C 180,E1 22053.839,E2 22053.839} C_VEL
LIN {X 0,Y 447.978,Z 773.859,A -85,B 0,C 180,E1 22051.279,E2 22051.279} C_VEL
LIN {X 0,Y 448.004,Z 772.099,A -85,B 0,C 180,E1 22048.721,E2 22048.721} C_VEL
LIN {X 0,Y 448.091,Z 768.721,A -85,B 0,C 180,E1 22046.162,E2 22046.162} C_VEL
LIN {X 0,Y 448.292,Z 763.722,A -85,B 0,C 180,E1 22043.597,E2 22043.597} C_VEL
LIN {X 0,Y 448.679,Z 756.974,A -85,B 0,C 180,E1 22041.026,E2 22041.026} C_VEL
LIN {X 0,Y 449.291,Z 748.79,A -85,B 0,C 180,E1 22038.576,E2 22038.576} C_VEL
LIN {X 0,Y 450.14,Z 739.239,A -85,B 0,C 180,E1 22036.251,E2 22036.251} C_VEL
LIN {X 0,Y 451.305,Z 727.632,A -85,B 0,C 180,E1 22033.923,E2 22033.923} C_VEL
LIN {X 0,Y 452.734,Z 714.438,A -85,B 0,C 180,E1 22031.723,E2 22031.723} C_VEL
LIN {X 0,Y 454.391,Z 699.595,A -85,B 0,C 180,E1 22029.655,E2 22029.655} C_VEL
LIN {X 0,Y 456.166,Z 683.564,A -85,B 0,C 180,E1 22027.784,E2 22027.784} C_VEL
LIN {X 0,Y 458.018,Z 666.463,A -85,B 0,C 180,E1 22026.112,E2 22026.112} C_VEL
LIN {X 0,Y 459.842,Z 648.331,A -85,B 0,C 180,E1 22024.637,E2 22024.637} C_VEL
LIN {X 0,Y 461.486,Z 630.166,A -85,B 0,C 180,E1 22023.423,E2 22023.423} C_VEL
LIN {X 0,Y 462.98,Z 611.319,A -85,B 0,C 180,E1 22022.404,E2 22022.404} C_VEL
LIN {X 0,Y 464.28,Z 591.039,A -85,B 0,C 180,E1 22021.553,E2 22021.553} C_VEL
LIN {X 0,Y 465.293,Z 570.014,A -85,B 0,C 180,E1 22020.918,E2 22020.918} C_VEL
LIN {X 0,Y 469.583,Z 462.245,A -85,B 0,C 180,E1 22018.69,E2 22018.69} C_VEL
LIN {X 0,Y 472.415,Z 376.277,A -85,B 0,C 180,E1 22017.106,E2 22017.106} C_VEL
LIN {X 0,Y 473.386,Z 326.711,A -85,B 0,C 180,E1 22016.257,E2 22016.257} C_VEL
LIN {X 0,Y 473.175,Z 324.703,A -85,B 0,C 180,E1 22016.145,E2 22016.145} C_VEL
LIN {X 0,Y 474.558,Z 309.552,A -85,B 0,C 180,E1 22014.739,E2 22014.739} C_VEL
LIN {X 0,Y 466.599,Z 291.765,A -85,B 0,C 180,E1 22011.656,E2 22011.656} C_VEL
LIN {X 0,Y 459.844,Z 277.989,A -85,B 0,C 180,E1 22008.982,E2 22008.982} C_VEL
LIN {X 0,Y 455.779,Z 270.046,A -85,B 0,C 180,E1 22007.323,E2 22007.323} C_VEL
LIN {X 0,Y 453.492,Z 265.646,A -85,B 0,C 180,E1 22006.361,E2 22006.361} C_VEL
LIN {X 0,Y 451.206,Z 261.255,A -85,B 0,C 180,E1 22005.375,E2 22005.375} C_VEL
LIN {X 0,Y 449.385,Z 258.01,A -85,B 0,C 180,E1 22004.603,E2 22004.603} C_VEL
LIN {X 0,Y 449.141,Z 256.792,A -85,B 0,C 180,E1 22004.349,E2 22004.349} C_VEL
LIN {X 0,Y 449.131,Z 256.77,A -85,B 0,C 180,E1 22000.546,E2 22000.546} C_VEL
LIN {X 0,Y 449.116,Z 256.77,A -85,B 0,C 180,E1 21996.942,E2 21996.942} C_VEL
LIN {X 0,Y 449.119,Z 256.793,A -85,B 0,C 180,E1 21993.36,E2 21993.36} C_VEL
LIN {X 0,Y 449.15,Z 256.971,A -85,B 0,C 180,E1 21992.959,E2 21992.959} C_VEL
LIN {X 0,Y 457.688,Z 282.801,A -85,B 0,C 180,E1 21990.106,E2 21990.106} C_VEL
LIN {X 0,Y 458.851,Z 287.12,A -85,B 0,C 180,E1 21989.647,E2 21989.647} C_VEL
LIN {X 0,Y 457.93,Z 329.406,A -85,B 0,C 180,E1 21986.032,E2 21986.032} C_VEL
LIN {X 0,Y 456.866,Z 370.489,A -85,B 0,C 180,E1 21982.52,E2 21982.52} C_VEL
LIN {X 0,Y 455.643,Z 413.973,A -85,B 0,C 180,E1 21978.819,E2 21978.819} C_VEL
LIN {X 0,Y 454.673,Z 450.352,A -85,B 0,C 180,E1 21975.75,E2 21975.75} C_VEL
LIN {X 0,Y 453.018,Z 594.269,A -85,B 0,C 180,E1 21973.185,E2 21973.185} C_VEL
LIN {X 0,Y 452.849,Z 610.767,A -85,B 0,C 180,E1 21972.659,E2 21972.659} C_VEL
LIN {X 0,Y 452.496,Z 626.309,A -85,B 0,C 180,E1 21971.924,E2 21971.924} C_VEL
LIN {X 0,Y 452.051,Z 641.451,A -85,B 0,C 180,E1 21970.966,E2 21970.966} C_VEL
LIN {X 0,Y 451.517,Z 655.711,A -85,B 0,C 180,E1 21969.791,E2 21969.791} C_VEL
LIN {X 0,Y 450.98,Z 668.377,A -85,B 0,C 180,E1 21968.479,E2 21968.479} C_VEL
LIN {X 0,Y 450.426,Z 680.662,A -85,B 0,C 180,E1 21966.885,E2 21966.885} C_VEL
LIN {X 0,Y 449.958,Z 690.764,A -85,B 0,C 180,E1 21965.228,E2 21965.228} C_VEL
LIN {X 0,Y 449.608,Z 699.409,A -85,B 0,C 180,E1 21963.443,E2 21963.443} C_VEL
LIN {X 0,Y 449.353,Z 706.448,A -85,B 0,C 180,E1 21961.531,E2 21961.531} C_VEL
LIN {X 0,Y 449.205,Z 711.617,A -85,B 0,C 180,E1 21959.618,E2 21959.618} C_VEL
LIN {X 0,Y 449.134,Z 715.378,A -85,B 0,C 180,E1 21957.449,E2 21957.449} C_VEL
LIN {X 0,Y 449.144,Z 716.999,A -85,B 0,C 180,E1 21955.404,E2 21955.404} C_VEL
LIN {X 0,Y 449.224,Z 716.851,A -85,B 0,C 180,E1 21953.354,E2 21953.354} C_VEL
LIN {X 0,Y 449.357,Z 714.781,A -85,B 0,C 180,E1 21951.298,E2 21951.298} C_VEL
LIN {X 0,Y 449.581,Z 711.108,A -85,B 0,C 180,E1 21949.363,E2 21949.363} C_VEL
LIN {X 0,Y 449.87,Z 705.231,A -85,B 0,C 180,E1 21947.345,E2 21947.345} C_VEL
LIN {X 0,Y 450.236,Z 698.253,A -85,B 0,C 180,E1 21945.598,E2 21945.598} C_VEL
LIN {X 0,Y 450.698,Z 689.266,A -85,B 0,C 180,E1 21943.864,E2 21943.864} C_VEL
LIN {X 0,Y 451.19,Z 679.099,A -85,B 0,C 180,E1 21942.327,E2 21942.327} C_VEL
LIN {X 0,Y 451.727,Z 667.04,A -85,B 0,C 180,E1 21940.878,E2 21940.878} C_VEL
LIN {X 0,Y 452.179,Z 653.932,A -85,B 0,C 180,E1 21939.645,E2 21939.645} C_VEL
LIN {X 0,Y 452.564,Z 640.075,A -85,B 0,C 180,E1 21938.621,E2 21938.621} C_VEL
LIN {X 0,Y 452.838,Z 624.245,A -85,B 0,C 180,E1 21937.742,E2 21937.742} C_VEL
LIN {X 0,Y 452.956,Z 608.252,A -85,B 0,C 180,E1 21937.122,E2 21937.122} C_VEL
LIN {X 0,Y 452.9,Z 591.506,A -85,B 0,C 180,E1 21936.717,E2 21936.717} C_VEL
LIN {X 0,Y 454.058,Z 503.52,A -85,B 0,C 180,E1 21935.131,E2 21935.131} C_VEL
LIN {X 0,Y 454.999,Z 460.77,A -85,B 0,C 180,E1 21934.279,E2 21934.279} C_VEL
LIN {X 0,Y 456.319,Z 453.043,A -85,B 0,C 180,E1 21933.73,E2 21933.73} C_VEL
LIN {X 0,Y 456.998,Z 411.759,A -85,B 0,C 180,E1 21930.438,E2 21930.438} C_VEL
LIN {X 0,Y 457.315,Z 377.993,A -85,B 0,C 180,E1 21927.827,E2 21927.827} C_VEL
LIN {X 0,Y 457.428,Z 349.43,A -85,B 0,C 180,E1 21925.672,E2 21925.672} C_VEL
LIN {X 0,Y 459.323,Z 350.01,A -85,B 0,C 180,E1 21925.379,E2 21925.379} C_VEL
LIN {X 0,Y 461.951,Z 349.294,A -85,B 0,C 180,E1 21925.117,E2 21925.117} C_VEL
LIN {X 0,Y 463.543,Z 348.558,A -85,B 0,C 180,E1 21924.988,E2 21924.988} C_VEL
LIN {X 0,Y 467.586,Z 347.873,A -85,B 0,C 180,E1 21924.559,E2 21924.559} C_VEL
LIN {X 0,Y 470.306,Z 347.084,A -85,B 0,C 180,E1 21924.304,E2 21924.304} C_VEL
LIN {X 0,Y 476.762,Z 345.62,A -85,B 0,C 180,E1 21923.682,E2 21923.682} C_VEL
LIN {X 0,Y 476.736,Z 363.805,A -85,B 0,C 180,E1 21922.16,E2 21922.16} C_VEL
LIN {X 0,Y 478.563,Z 380.964,A -85,B 0,C 180,E1 21920.57,E2 21920.57} C_VEL
LIN {X 0,Y 482.171,Z 396.173,A -85,B 0,C 180,E1 21919.009,E2 21919.009} C_VEL
LIN {X 0,Y 487.291,Z 409.103,A -85,B 0,C 180,E1 21917.541,E2 21917.541} C_VEL
LIN {X 0,Y 494.197,Z 420.963,A -85,B 0,C 180,E1 21916.056,E2 21916.056} C_VEL
LIN {X 0,Y 503.114,Z 431.745,A -85,B 0,C 180,E1 21914.55,E2 21914.55} C_VEL
LIN {X 0,Y 512.916,Z 440.298,A -85,B 0,C 180,E1 21913.193,E2 21913.193} C_VEL
LIN {X 0,Y 523.967,Z 447.34,A -85,B 0,C 180,E1 21911.909,E2 21911.909} C_VEL
LIN {X 0,Y 527.575,Z 449.415,A -85,B 0,C 180,E1 21911.52,E2 21911.52} C_VEL
LIN {X 0,Y 508.605,Z 478.558,A -85,B 0,C 180,E1 21910.893,E2 21910.893} C_VEL
LIN {X 0,Y 498.554,Z 496.42,A -85,B 0,C 180,E1 21910.375,E2 21910.375} C_VEL
LIN {X 0,Y 491.762,Z 511.194,A -85,B 0,C 180,E1 21909.827,E2 21909.827} C_VEL
LIN {X 0,Y 482.43,Z 530.373,A -85,B 0,C 180,E1 21909.131,E2 21909.131} C_VEL
LIN {X 0,Y 473.543,Z 554.324,A -85,B 0,C 180,E1 21908.081,E2 21908.081} C_VEL
LIN {X 0,Y 472.15,Z 572.487,A -85,B 0,C 180,E1 21907.865,E2 21907.865} C_VEL
LIN {X 0,Y 471.244,Z 602.706,A -85,B 0,C 180,E1 21907.309,E2 21907.309} C_VEL
LIN {X 0,Y 469.724,Z 626.71,A -85,B 0,C 180,E1 21906.661,E2 21906.661} C_VEL
LIN {X 0,Y 468.04,Z 649.221,A -85,B 0,C 180,E1 21905.827,E2 21905.827} C_VEL
LIN {X 0,Y 466.126,Z 671.131,A -85,B 0,C 180,E1 21904.791,E2 21904.791} C_VEL
LIN {X 0,Y 464.208,Z 691.322,A -85,B 0,C 180,E1 21903.611,E2 21903.611} C_VEL
LIN {X 0,Y 462.03,Z 711.866,A -85,B 0,C 180,E1 21902.165,E2 21902.165} C_VEL
LIN {X 0,Y 459.833,Z 731.462,A -85,B 0,C 180,E1 21900.512,E2 21900.512} C_VEL
LIN {X 0,Y 457.697,Z 749.327,A -85,B 0,C 180,E1 21898.725,E2 21898.725} C_VEL
LIN {X 0,Y 455.588,Z 766.796,A -85,B 0,C 180,E1 21896.667,E2 21896.667} C_VEL
LIN {X 0,Y 453.584,Z 783.495,A -85,B 0,C 180,E1 21894.344,E2 21894.344} C_VEL
LIN {X 0,Y 451.918,Z 798.015,A -85,B 0,C 180,E1 21891.957,E2 21891.957} C_VEL
LIN {X 0,Y 450.689,Z 809.724,A -85,B 0,C 180,E1 21889.707,E2 21889.707} C_VEL
LIN {X 0,Y 449.524,Z 821.407,A -85,B 0,C 180,E1 21886.941,E2 21886.941} C_VEL
LIN {X 0,Y 448.723,Z 831.352,A -85,B 0,C 180,E1 21884.056,E2 21884.056} C_VEL
LIN {X 0,Y 448.248,Z 839.213,A -85,B 0,C 180,E1 21881.19,E2 21881.19} C_VEL
LIN {X 0,Y 448.03,Z 845.152,A -85,B 0,C 180,E1 21878.341,E2 21878.341} C_VEL
LIN {X 0,Y 447.936,Z 849.134,A -85,B 0,C 180,E1 21875.636,E2 21875.636} C_VEL
LIN {X 0,Y 447.913,Z 851.577,A -85,B 0,C 180,E1 21872.943,E2 21872.943} C_VEL
LIN {X 0,Y 447.909,Z 852.489,A -85,B 0,C 180,E1 21870.128,E2 21870.128} C_VEL
LIN {X 0,Y 447.908,Z 851.784,A -85,B 0,C 180,E1 21867.441,E2 21867.441} C_VEL
LIN {X 0,Y 447.931,Z 849.592,A -85,B 0,C 180,E1 21864.749,E2 21864.749} C_VEL
LIN {X 0,Y 448.015,Z 845.601,A -85,B 0,C 180,E1 21861.917,E2 21861.917} C_VEL
LIN {X 0,Y 448.222,Z 839.813,A -85,B 0,C 180,E1 21859.07,E2 21859.07} C_VEL
LIN {X 0,Y 448.636,Z 832.521,A -85,B 0,C 180,E1 21856.334,E2 21856.334} C_VEL
LIN {X 0,Y 449.308,Z 823.853,A -85,B 0,C 180,E1 21853.716,E2 21853.716} C_VEL
LIN {X 0,Y 450.377,Z 812.717,A -85,B 0,C 180,E1 21850.953,E2 21850.953} C_VEL
LIN {X 0,Y 451.52,Z 801.663,A -85,B 0,C 180,E1 21848.705,E2 21848.705} C_VEL
LIN {X 0,Y 453.077,Z 787.754,A -85,B 0,C 180,E1 21846.319,E2 21846.319} C_VEL
LIN {X 0,Y 454.957,Z 771.887,A -85,B 0,C 180,E1 21844.008,E2 21844.008} C_VEL
LIN {X 0,Y 457.123,Z 754.038,A -85,B 0,C 180,E1 21841.806,E2 21841.806} C_VEL
LIN {X 0,Y 459.222,Z 736.201,A -85,B 0,C 180,E1 21839.948,E2 21839.948} C_VEL
LIN {X 0,Y 461.472,Z 716.701,A -85,B 0,C 180,E1 21838.23,E2 21838.23} C_VEL
LIN {X 0,Y 463.613,Z 696.255,A -85,B 0,C 180,E1 21836.73,E2 21836.73} C_VEL
LIN {X 0,Y 465.663,Z 675.647,A -85,B 0,C 180,E1 21835.468,E2 21835.468} C_VEL
LIN {X 0,Y 467.685,Z 652.542,A -85,B 0,C 180,E1 21834.33,E2 21834.33} C_VEL
LIN {X 0,Y 469.456,Z 629.445,A -85,B 0,C 180,E1 21833.448,E2 21833.448} C_VEL
LIN {X 0,Y 470.947,Z 605.729,A -85,B 0,C 180,E1 21832.784,E2 21832.784} C_VEL
LIN {X 0,Y 471.899,Z 580.63,A -85,B 0,C 180,E1 21832.287,E2 21832.287} C_VEL
LIN {X 0,Y 472.565,Z 564.715,A -85,B 0,C 180,E1 21832.052,E2 21832.052} C_VEL
LIN {X 0,Y 473.826,Z 554.166,A -85,B 0,C 180,E1 21831.962,E2 21831.962} C_VEL
LIN {X 0,Y 483.903,Z 532.624,A -85,B 0,C 180,E1 21830.858,E2 21830.858} C_VEL
LIN {X 0,Y 492.219,Z 518.871,A -85,B 0,C 180,E1 21830.293,E2 21830.293} C_VEL
LIN {X 0,Y 495.495,Z 513.529,A -85,B 0,C 180,E1 21830.081,E2 21830.081} C_VEL
LIN {X 0,Y 503.774,Z 499.727,A -85,B 0,C 180,E1 21829.533,E2 21829.533} C_VEL
LIN {X 0,Y 515.518,Z 483.501,A -85,B 0,C 180,E1 21829.037,E2 21829.037} C_VEL
LIN {X 0,Y 518.303,Z 479.778,A -85,B 0,C 180,E1 21828.933,E2 21828.933} C_VEL
LIN {X 0,Y 507.263,Z 472.779,A -85,B 0,C 180,E1 21827.659,E2 21827.659} C_VEL
LIN {X 0,Y 497.142,Z 464.01,A -85,B 0,C 180,E1 21826.221,E2 21826.221} C_VEL
LIN {X 0,Y 488.821,Z 453.967,A -85,B 0,C 180,E1 21824.719,E2 21824.719} C_VEL
LIN {X 0,Y 482.687,Z 443.541,A -85,B 0,C 180,E1 21823.286,E2 21823.286} C_VEL
LIN {X 0,Y 477.766,Z 431.17,A -85,B 0,C 180,E1 21821.721,E2 21821.721} C_VEL
LIN {X 0,Y 474.413,Z 416.248,A -85,B 0,C 180,E1 21820.001,E2 21820.001} C_VEL
LIN {X 0,Y 473.031,Z 399.733,A -85,B 0,C 180,E1 21818.266,E2 21818.266} C_VEL
LIN {X 0,Y 473.72,Z 380.851,A -85,B 0,C 180,E1 21816.47,E2 21816.47} C_VEL
LIN {X 0,Y 478.588,Z 337.309,A -85,B 0,C 180,E1 21812.545,E2 21812.545} C_VEL
LIN {X 0,Y 480.602,Z 319.95,A -85,B 0,C 180,E1 21810.921,E2 21810.921} C_VEL
LIN {X 0,Y 477.075,Z 311.95,A -85,B 0,C 180,E1 21809.506,E2 21809.506} C_VEL
LIN {X 0,Y 467.841,Z 315.084,A -85,B 0,C 180,E1 21808.463,E2 21808.463} C_VEL
LIN {X 0,Y 462.496,Z 316.976,A -85,B 0,C 180,E1 21807.837,E2 21807.837} C_VEL
LIN {X 0,Y 461.405,Z 317.294,A -85,B 0,C 180,E1 21807.698,E2 21807.698} C_VEL
LIN {X 0,Y 458.162,Z 318.808,A -85,B 0,C 180,E1 21807.35,E2 21807.35} C_VEL
LIN {X 0,Y 456.236,Z 318.641,A -85,B 0,C 180,E1 21806.995,E2 21806.995} C_VEL
LIN {X 0,Y 456.318,Z 362.952,A -85,B 0,C 180,E1 21803.913,E2 21803.913} C_VEL
LIN {X 0,Y 455.899,Z 412.408,A -85,B 0,C 180,E1 21800.341,E2 21800.341} C_VEL
LIN {X 0,Y 455.152,Z 459.268,A -85,B 0,C 180,E1 21796.856,E2 21796.856} C_VEL
LIN {X 0,Y 454.203,Z 500.933,A -85,B 0,C 180,E1 21793.688,E2 21793.688} C_VEL
LIN {X 0,Y 453.187,Z 507.898,A -85,B 0,C 180,E1 21793.246,E2 21793.246} C_VEL
LIN {X 0,Y 451.904,Z 611.646,A -85,B 0,C 180,E1 21791.374,E2 21791.374} C_VEL
LIN {X 0,Y 451.967,Z 627.235,A -85,B 0,C 180,E1 21790.987,E2 21790.987} C_VEL
LIN {X 0,Y 451.893,Z 642.105,A -85,B 0,C 180,E1 21790.367,E2 21790.367} C_VEL
LIN {X 0,Y 451.644,Z 656.197,A -85,B 0,C 180,E1 21789.517,E2 21789.517} C_VEL
LIN {X 0,Y 451.312,Z 669.297,A -85,B 0,C 180,E1 21788.444,E2 21788.444} C_VEL
LIN {X 0,Y 450.931,Z 680.408,A -85,B 0,C 180,E1 21787.26,E2 21787.26} C_VEL
LIN {X 0,Y 450.553,Z 689.883,A -85,B 0,C 180,E1 21785.986,E2 21785.986} C_VEL
LIN {X 0,Y 450.159,Z 698.74,A -85,B 0,C 180,E1 21784.458,E2 21784.458} C_VEL
LIN {X 0,Y 449.809,Z 706.007,A -85,B 0,C 180,E1 21782.803,E2 21782.803} C_VEL
LIN {X 0,Y 449.544,Z 711.337,A -85,B 0,C 180,E1 21781.147,E2 21781.147} C_VEL
LIN {X 0,Y 449.351,Z 715.202,A -85,B 0,C 180,E1 21779.362,E2 21779.362} C_VEL
LIN {X 0,Y 449.217,Z 717.353,A -85,B 0,C 180,E1 21777.448,E2 21777.448} C_VEL
LIN {X 0,Y 449.154,Z 717.628,A -85,B 0,C 180,E1 21775.659,E2 21775.659} C_VEL
LIN {X 0,Y 449.15,Z 716.266,A -85,B 0,C 180,E1 21773.866,E2 21773.866} C_VEL
LIN {X 0,Y 449.213,Z 712.899,A -85,B 0,C 180,E1 21771.939,E2 21771.939} C_VEL
LIN {X 0,Y 449.358,Z 707.832,A -85,B 0,C 180,E1 21770.134,E2 21770.134} C_VEL
LIN {X 0,Y 449.582,Z 701.238,A -85,B 0,C 180,E1 21768.453,E2 21768.453} C_VEL
LIN {X 0,Y 449.897,Z 693.243,A -85,B 0,C 180,E1 21766.897,E2 21766.897} C_VEL
LIN {X 0,Y 450.289,Z 682.86,A -85,B 0,C 180,E1 21765.336,E2 21765.336} C_VEL
LIN {X 0,Y 450.714,Z 671.087,A -85,B 0,C 180,E1 21763.967,E2 21763.967} C_VEL
LIN {X 0,Y 451.106,Z 658.157,A -85,B 0,C 180,E1 21762.805,E2 21762.805} C_VEL
LIN {X 0,Y 451.46,Z 644.408,A -85,B 0,C 180,E1 21761.87,E2 21761.87} C_VEL
LIN {X 0,Y 451.68,Z 630.071,A -85,B 0,C 180,E1 21761.16,E2 21761.16} C_VEL
LIN {X 0,Y 451.787,Z 615.138,A -85,B 0,C 180,E1 21760.67,E2 21760.67} C_VEL
LIN {X 0,Y 452.997,Z 499.762,A -85,B 0,C 180,E1 21758.642,E2 21758.642} C_VEL
LIN {X 0,Y 454.138,Z 460.504,A -85,B 0,C 180,E1 21755.549,E2 21755.549} C_VEL
LIN {X 0,Y 455.428,Z 412.67,A -85,B 0,C 180,E1 21751.763,E2 21751.763} C_VEL
LIN {X 0,Y 456.601,Z 367.041,A -85,B 0,C 180,E1 21748.147,E2 21748.147} C_VEL
LIN {X 0,Y 457.633,Z 323.642,A -85,B 0,C 180,E1 21744.697,E2 21744.697} C_VEL
LIN {X 0,Y 458.451,Z 285.096,A -85,B 0,C 180,E1 21741.634,E2 21741.634} C_VEL
LIN {X 0,Y 455.511,Z 275.583,A -85,B 0,C 180,E1 21740.627,E2 21740.627} C_VEL
LIN {X 0,Y 457.46,Z 275.724,A -85,B 0,C 180,E1 21740.177,E2 21740.177} C_VEL
LIN {X 0,Y 458.945,Z 275.841,A -85,B 0,C 180,E1 21739.844,E2 21739.844} C_VEL
LIN {X 0,Y 463.762,Z 286.131,A -85,B 0,C 180,E1 21737.223,E2 21737.223} C_VEL
LIN {X 0,Y 468.938,Z 297.393,A -85,B 0,C 180,E1 21734.589,E2 21734.589} C_VEL
LIN {X 0,Y 474.602,Z 311.09,A -85,B 0,C 180,E1 21731.739,E2 21731.739} C_VEL
LIN {X 0,Y 474.971,Z 312.738,A -85,B 0,C 180,E1 21731.46,E2 21731.46} C_VEL
LIN {X 0,Y 474.332,Z 317.342,A -85,B 0,C 180,E1 21730.942,E2 21730.942} C_VEL
LIN {X 0,Y 473.491,Z 321.795,A -85,B 0,C 180,E1 21730.565,E2 21730.565} C_VEL
LIN {X 0,Y 471.68,Z 328.892,A -85,B 0,C 180,E1 21730.246,E2 21730.246} C_VEL
LIN {X 0,Y 468.884,Z 339.874,A -85,B 0,C 180,E1 21730.057,E2 21730.057} C_VEL
LIN {X 0,Y 467.395,Z 350.141,A -85,B 0,C 180,E1 21729.946,E2 21729.946} C_VEL
LIN {X 0,Y 467.35,Z 351.287,A -85,B 0,C 180,E1 21729.928,E2 21729.928} C_VEL
LIN {X 0,Y 464.942,Z 428.668,A -85,B 0,C 180,E1 21728.539,E2 21728.539} C_VEL
LIN {X 0,Y 460.939,Z 522.171,A -85,B 0,C 180,E1 21726.632,E2 21726.632} C_VEL
LIN {X 0,Y 458.444,Z 577.303,A -85,B 0,C 180,E1 21725.38,E2 21725.38} C_VEL
LIN {X 0,Y 457.258,Z 597.816,A -85,B 0,C 180,E1 21724.674,E2 21724.674} C_VEL
LIN {X 0,Y 455.769,Z 617.679,A -85,B 0,C 180,E1 21723.752,E2 21723.752} C_VEL
LIN {X 0,Y 454.088,Z 636.343,A -85,B 0,C 180,E1 21722.648,E2 21722.648} C_VEL
LIN {X 0,Y 452.184,Z 654.755,A -85,B 0,C 180,E1 21721.308,E2 21721.308} C_VEL
LIN {X 0,Y 450.309,Z 671.599,A -85,B 0,C 180,E1 21719.826,E2 21719.826} C_VEL
LIN {X 0,Y 448.253,Z 688.929,A -85,B 0,C 180,E1 21718.004,E2 21718.004} C_VEL
LIN {X 0,Y 446.357,Z 704.544,A -85,B 0,C 180,E1 21716.043,E2 21716.043} C_VEL
LIN {X 0,Y 444.637,Z 719.043,A -85,B 0,C 180,E1 21713.877,E2 21713.877} C_VEL
LIN {X 0,Y 443.182,Z 731.94,A -85,B 0,C 180,E1 21711.577,E2 21711.577} C_VEL
LIN {X 0,Y 442.021,Z 743.218,A -85,B 0,C 180,E1 21709.147,E2 21709.147} C_VEL
LIN {X 0,Y 441.189,Z 752.425,A -85,B 0,C 180,E1 21706.728,E2 21706.728} C_VEL
LIN {X 0,Y 440.638,Z 759.853,A -85,B 0,C 180,E1 21704.32,E2 21704.32} C_VEL
LIN {X 0,Y 440.284,Z 766.201,A -85,B 0,C 180,E1 21701.661,E2 21701.661} C_VEL
LIN {X 0,Y 440.106,Z 770.704,A -85,B 0,C 180,E1 21699.019,E2 21699.019} C_VEL
LIN {X 0,Y 440.029,Z 773.538,A -85,B 0,C 180,E1 21696.393,E2 21696.393} C_VEL
LIN {X 0,Y 440.01,Z 774.801,A -85,B 0,C 180,E1 21693.779,E2 21693.779} C_VEL
LIN {X 0,Y 440.011,Z 774.532,A -85,B 0,C 180,E1 21691.172,E2 21691.172} C_VEL
LIN {X 0,Y 440.045,Z 772.73,A -85,B 0,C 180,E1 21688.568,E2 21688.568} C_VEL
LIN {X 0,Y 440.15,Z 769.28,A -85,B 0,C 180,E1 21685.962,E2 21685.962} C_VEL
LIN {X 0,Y 440.378,Z 764.191,A -85,B 0,C 180,E1 21683.351,E2 21683.351} C_VEL
LIN {X 0,Y 440.804,Z 757.336,A -85,B 0,C 180,E1 21680.732,E2 21680.732} C_VEL
LIN {X 0,Y 441.521,Z 748.526,A -85,B 0,C 180,E1 21678.107,E2 21678.107} C_VEL
LIN {X 0,Y 442.522,Z 738.099,A -85,B 0,C 180,E1 21675.609,E2 21675.609} C_VEL
LIN {X 0,Y 443.741,Z 726.812,A -85,B 0,C 180,E1 21673.372,E2 21673.372} C_VEL
LIN {X 0,Y 445.205,Z 714.191,A -85,B 0,C 180,E1 21671.267,E2 21671.267} C_VEL
LIN {X 0,Y 446.91,Z 699.945,A -85,B 0,C 180,E1 21669.259,E2 21669.259} C_VEL
LIN {X 0,Y 448.839,Z 683.685,A -85,B 0,C 180,E1 21667.332,E2 21667.332} C_VEL
LIN {X 0,Y 450.811,Z 666.566,A -85,B 0,C 180,E1 21665.636,E2 21665.636} C_VEL
LIN {X 0,Y 452.76,Z 648.388,A -85,B 0,C 180,E1 21664.141,E2 21664.141} C_VEL
LIN {X 0,Y 454.594,Z 629.118,A -85,B 0,C 180,E1 21662.846,E2 21662.846} C_VEL
LIN {X 0,Y 456.196,Z 609.719,A -85,B 0,C 180,E1 21661.808,E2 21661.808} C_VEL
LIN {X 0,Y 457.507,Z 589.554,A -85,B 0,C 180,E1 21660.976,E2 21660.976} C_VEL
LIN {X 0,Y 458.505,Z 569.313,A -85,B 0,C 180,E1 21660.378,E2 21660.378} C_VEL
LIN {X 0,Y 463.01,Z 464.828,A -85,B 0,C 180,E1 21658.159,E2 21658.159} C_VEL
LIN {X 0,Y 465.957,Z 381.73,A -85,B 0,C 180,E1 21656.598,E2 21656.598} C_VEL
LIN {X 0,Y 467.115,Z 328.4,A -85,B 0,C 180,E1 21655.674,E2 21655.674} C_VEL
LIN {X 0,Y 467.126,Z 326.012,A -85,B 0,C 180,E1 21655.495,E2 21655.495} C_VEL
LIN {X 0,Y 468.305,Z 313.741,A -85,B 0,C 180,E1 21654.347,E2 21654.347} C_VEL
LIN {X 0,Y 460.791,Z 296.809,A -85,B 0,C 180,E1 21651.367,E2 21651.367} C_VEL
LIN {X 0,Y 453.106,Z 280.808,A -85,B 0,C 180,E1 21648.209,E2 21648.209} C_VEL
LIN {X 0,Y 448.109,Z 271.293,A -85,B 0,C 180,E1 21646.114,E2 21646.114} C_VEL
LIN {X 0,Y 445.848,Z 267.007,A -85,B 0,C 180,E1 21645.127,E2 21645.127} C_VEL
LIN {X 0,Y 443.985,Z 263.284,A -85,B 0,C 180,E1 21644.263,E2 21644.263} C_VEL
LIN {X 0,Y 441.439,Z 259.015,A -85,B 0,C 180,E1 21643.16,E2 21643.16} C_VEL
LIN {X 0,Y 441.178,Z 257.78,A -85,B 0,C 180,E1 21642.891,E2 21642.891} C_VEL
LIN {X 0,Y 441.177,Z 257.778,A -85,B 0,C 180,E1 21639.222,E2 21639.222} C_VEL
LIN {X 0,Y 441.188,Z 257.771,A -85,B 0,C 180,E1 21635.463,E2 21635.463} C_VEL
LIN {X 0,Y 441.2,Z 257.917,A -85,B 0,C 180,E1 21633.454,E2 21633.454} C_VEL
LIN {X 0,Y 450.083,Z 284.556,A -85,B 0,C 180,E1 21630.464,E2 21630.464} C_VEL
LIN {X 0,Y 451.497,Z 290.05,A -85,B 0,C 180,E1 21629.886,E2 21629.886} C_VEL
LIN {X 0,Y 450.46,Z 332.58,A -85,B 0,C 180,E1 21626.213,E2 21626.213} C_VEL
LIN {X 0,Y 449.363,Z 373.407,A -85,B 0,C 180,E1 21622.709,E2 21622.709} C_VEL
LIN {X 0,Y 448.068,Z 416.459,A -85,B 0,C 180,E1 21619.014,E2 21619.014} C_VEL
LIN {X 0,Y 447.11,Z 451.396,A -85,B 0,C 180,E1 21616.056,E2 21616.056} C_VEL
LIN {X 0,Y 445.283,Z 595.272,A -85,B 0,C 180,E1 21613.427,E2 21613.427} C_VEL
LIN {X 0,Y 445.102,Z 612.006,A -85,B 0,C 180,E1 21612.883,E2 21612.883} C_VEL
LIN {X 0,Y 444.738,Z 627.534,A -85,B 0,C 180,E1 21612.135,E2 21612.135} C_VEL
LIN {X 0,Y 444.274,Z 642.694,A -85,B 0,C 180,E1 21611.16,E2 21611.16} C_VEL
LIN {X 0,Y 443.705,Z 657.389,A -85,B 0,C 180,E1 21609.927,E2 21609.927} C_VEL
LIN {X 0,Y 443.136,Z 670.22,A -85,B 0,C 180,E1 21608.565,E2 21608.565} C_VEL
LIN {X 0,Y 442.587,Z 682.007,A -85,B 0,C 180,E1 21607.008,E2 21607.008} C_VEL
LIN {X 0,Y 442.1,Z 692.128,A -85,B 0,C 180,E1 21605.321,E2 21605.321} C_VEL
LIN {X 0,Y 441.735,Z 700.796,A -85,B 0,C 180,E1 21603.504,E2 21603.504} C_VEL
LIN {X 0,Y 441.459,Z 708.277,A -85,B 0,C 180,E1 21601.428,E2 21601.428} C_VEL
